(* CoDeSys 2.3 project: cy-wg-017-01.pro *)
(* Title: cy-wg-06 - ClevergyAS *)
(* Author: Andrea Ravasio *)
(* Libraries: Standard.lib 2.12.10 14:48:34, Util.lib 26.9.14 10:12:46, Visual.lib 2.12.10 14:48:34, WagoLibIdent.lib 25.2.13 11:12:16, WagoLibStatus.lib 2.12.10 14:48:32, SysLibFile.lib 2.12.10 14:48:34, SysLibRtc.lib 2.12.10 14:48:32, SysLibSockets.lib 10.2.11 09:20:54, SysLibEvent.lib 2.12.10 14:48:34, SysLibPlcCtrl.lib 2.12.10 14:48:32, SysLibCallback.lib 2.12.10 14:48:32, mod_com.lib 2.12.10 14:48:32, SerComm.lib 31.5.11 08:54:36, Serial_Interface_01.lib 22.4.13 12:50:14, Modb_l05.lib 22.4.13 12:50:12, Ethernet.lib 2.12.10 14:48:32, MBus_03.lib 22.7.15 16:25:47, WagoLibModbus_IP_01.lib 24.7.13 15:05:58, WagoLibMBX_01.lib 20.3.12 16:32:40, LON_01.lib 22.7.15 16:25:47 *)

(* PLC configuration (modules and I/O channels)
0750-9999/0545-0008 8 DO/DI Generic [Type_34_8_Channels] node 0, in %IB60 out %QB36 {INTTypePAAssignment = PLC; INTTypeModule = plugged}
  VPN_ST2 AT %IX30.0 [BOOLOnX_I] Ch_1 Digital input
  LAMP_AL AT %QX18.0 [BOOLOnX_Q] Ch_1 Digital output
  KEY_QE_ST AT %IX30.1 [BOOLOnX_I] Ch_2 Digital input
  CIR02_EN AT %QX18.1 [BOOLOnX_Q] Ch_2 Digital output
  CTL01_ST AT %IX30.2 [BOOLOnX_I] Ch_3 Digital input
  CIR01_EN AT %QX18.2 [BOOLOnX_Q] Ch_3 Digital output
  CTL02_ST AT %IX30.3 [BOOLOnX_I] Ch_4 Digital input
  AT %QX18.3 [BOOLOnX_Q] Ch_4 Digital output
  CIRD01_A_AL AT %IX30.4 [BOOLOnX_I] Ch_5 Digital input
  AT %QX18.4 [BOOLOnX_Q] Ch_5 Digital output
  CIRD01_A_AUTO AT %IX30.5 [BOOLOnX_I] Ch_6 Digital input
  AT %QX18.5 [BOOLOnX_Q] Ch_6 Digital output
  CIRD01_B_AL AT %IX30.6 [BOOLOnX_I] Ch_7 Digital input
  AT %QX18.6 [BOOLOnX_Q] Ch_7 Digital output
  CIRD01_B_AUTO AT %IX30.7 [BOOLOnX_I] Ch_8 Digital input
  AT %QX18.7 [BOOLOnX_Q] Ch_8 Digital output
0750-9999/0400-0008 8 DI Generic [Type_1_8_Channels] node 1, in %IB60 out %QB36 {INTTypePAAssignment = PLC; INTTypeModule = plugged}
  CIRD02_A_AL AT %IX30.8 [BOOLOnX_I] I 1: Digital Input
  CIR03_AL AT %IX30.9 [BOOLOnX_I] I 2: Digital Input
  CIRD02_A_AUTO AT %IX30.10 [BOOLOnX_I] I 3: Digital Input
  CIR03_AUTO AT %IX30.11 [BOOLOnX_I] I 4: Digital Input
  CIRD02_B_AL AT %IX30.12 [BOOLOnX_I] I 5: Digital Input
  CIR02_AL AT %IX30.13 [BOOLOnX_I] I 6: Digital Input
  CIRD02_B_AUTO AT %IX30.14 [BOOLOnX_I] I 7: Digital Input
  CIR02_ST AT %IX30.15 [BOOLOnX_I] I 8: Digital Input
0750-9999/0400-0004 4 DI Generic [Type_1_4_Channels] node 2, in %IB61 out %QB37 {INTTypePAAssignment = PLC; INTTypeModule = plugged}
  CIR02_AUTO AT %IX31.0 [BOOLOnX_I] I 1: Digital Input
  CIR01_ST AT %IX31.1 [BOOLOnX_I] I 2: Digital Input
  CIR01_AL AT %IX31.2 [BOOLOnX_I] I 3: Digital Input
  CIR01_AUTO AT %IX31.3 [BOOLOnX_I] I 4: Digital Input
0750-0478 2 AI 0-10V 16 Bit S.E. [Type_8_2_Channels] node 3, in %IB56 out %QB36 {INTTypePAAssignment = PLC; INTTypeModule = plugged}
  VRD04_ST AT %IW0 [WORDOnW_I] I 1: Analog Input
  VRD05_ST AT %IW1 [WORDOnW_I] I 2: Analog Input
0753-0648 LON-FTT [Type_55_1_Channels] node 4, in %IB56 out %QB36 {INTTypePAAssignment = PLC; INTTypeModule = plugged; DataStream = .; DataStream = .; DataStream = .; DataStream = .; DataStream = .; DataStream = .; DataStream = .; DataStream = .; DataStream = .; DataStream = .; DataStream = .; DataStream = .; DataStream = .; DataStream = .; DataStream = .; DataStream = .; DataStream = .; DataStream = .; DataStream = .; DataStream = .; DataStream = .; DataStream = .; DataStream = .; DataStream = .; DataStream = .; DataStream = .; DataStream = .; DataStream = .; DataStream = .; DataStream = .; DataStream = .; DataStream = .; DataStream = .; DataStream = .; DataStream = .; DataStream = .; DataStream = .; DataStream = .; DataStream = .; DataStream = .; DataStream = .; DataStream = .; DataStream = .; DataStream = .; DataStream = .; DataStream = .; DataStream = .; DataStream = .; DataStream = .; DataStream = .; DataStream = .; DataStream = .; DataStream = .; DataStream = .; DataStream = .; DataStream = .; DataStream = .; DataStream = .; DataStream = .; DataStream = .; DataStream = .; DataStream = .; DataStream = .; DataStream = .; DataStream = .; DataStream = .; DataStream = .; DataStream = .; DataStream = .; DataStream = .; DataStream = .; DataStream = .; DataStream = .; DataStream = .; DataStream = .; DataStream = .; DataStream = .; DataStream = .; DataStream = .; DataStream = .; DataStream = .; DataStream = .; DataStream = .; DataStream = .; DataStream = .; DataStream = .; DataStream = .; DataStream = .; DataStream = .; DataStream = .; DataStream = .; DataStream = .; DataStream = .; DataStream = .; DataStream = .; DataStream = .; DataStream = .; DataStream = .; DataStream = .; DataStream = .; DataStream = .; DataStream = .; DataStream = .; DataStream = .; DataStream = .; DataStream = .; DataStream = .; DataStream = .; DataStream = .; DataStream = .; DataStream = .; DataStream = .; DataStream = .; DataStream = .; DataStream = .; DataStream = .; DataStream = .; DataStream = .; DataStream = .; DataStream = .; DataStream = .; DataStream = .; DataStream = .; DataStream = .; DataStream = .; DataStream = .; DataStream = .; DataStream = .; DataStream = .; DataStream = .; DataStream = .; DataStream = .; DataStream = .; DataStream = .; DataStream = .; DataStream = .; DataStream = .; DataStream = .; DataStream = .; DataStream = .; DataStream = .; DataStream = .; DataStream = .; DataStream = .; DataStream = .; DataStream = .; DataStream = .; DataStream = .; DataStream = .; DataStream = .; DataStream = .; DataStream = .; DataStream = .; DataStream = .; DataStream = .; DataStream = .; DataStream = .; DataStream = .; DataStream = .; DataStream = .; DataStream = .; DataStream = .; DataStream = .; DataStream = .; DataStream = .; DataStream = .; DataStream = .; DataStream = .; DataStream = .; DataStream = .; DataStream = .; DataStream = .; DataStream = .; DataStream = .; DataStream = .; DataStream = .; DataStream = .; DataStream = .; DataStream = .; DataStream = .; DataStream = .; DataStream = .; DataStream = .; DataStream = .; DataStream = .; DataStream = .; DataStream = .; DataStream = .; DataStream = .; DataStream = .; DataStream = .; DataStream = .; DataStream = .; DataStream = .; DataStream = .; DataStream = .; DataStream = .; DataStream = .; DataStream = .; DataStream = .}
  AT %IB4 [BYTEOnB_I] First Byte of 24
  AT %QB0 [BYTEOnB_Q] First Byte of 24
0750-0464#04 2/4 AI RTD / ADJ./ HA [Type_44_4_Channels] node 5, in %IB60 out %QB36 {INTTypePAAssignment = PLC; INTTypeModule = plugged}
  S01 AT %IW14 [INTOnW_I] Channel 1
  S02 AT %IW15 [INTOnW_I] Channel 2
  S03 AT %IW16 [INTOnW_I] Channel 3
  S04 AT %IW17 [INTOnW_I] Channel 4
0750-0464#04 2/4 AI RTD / ADJ./ HA [Type_44_4_Channels] node 6, in %IB84 out %QB60 {INTTypePAAssignment = PLC; INTTypeModule = plugged}
  S05 AT %IW18 [INTOnW_I] Channel 1
  S07 AT %IW19 [INTOnW_I] Channel 2
  S06 AT %IW20 [INTOnW_I] Channel 3
  S08 AT %IW21 [INTOnW_I] Channel 4
0750-0556 2 AO ±10V [Type_14_2_Channels] node 7, in %IB92 out %QB60 {INTTypePAAssignment = PLC; INTTypeModule = plugged}
  VRD04_CTRL AT %QW12 [WORDOnW_Q] O 1: Analog Output
  VRD05_CTRL AT %QW13 [WORDOnW_Q] O 2: Analog Output
0750-0650/0003-0000#03 RS 232 C Interface (Adjustable), 3 Byte [Type_21_1_Channels] node 8, in %IB100 out %QB60 {INTTypePAAssignment = PLC; INTTypeModule = plugged}
  AT %IX22.0 [BOOLOnX_I] Transmission acknowledgement
  AT %IX22.1 [BOOLOnX_I] Reception request
  AT %IX22.2 [BOOLOnX_I] Initialization acknowledgement
  AT %IX22.3 [BOOLOnX_I] Input buffer is full
  AT %IX22.4 [BOOLOnX_I] Number of received characters Bit 0
  AT %IX22.5 [BOOLOnX_I] Number of received characters Bit 1
  AT %IX22.6 [BOOLOnX_I] Number of received characters Bit 2
  AT %IB45 [BYTEOnB_I] Input data Byte 0
  AT %IB46 [BYTEOnB_I] Input data Byte 1
  AT %IB47 [BYTEOnB_I] Input data Byte 2
  AT %QX14.0 [BOOLOnX_Q] Transmission request
  AT %QX14.1 [BOOLOnX_Q] Reception acknowledgement
  AT %QX14.2 [BOOLOnX_Q] Initialization request
  AT %QX14.4 [BOOLOnX_Q] Number of characters Bit 0
  AT %QX14.5 [BOOLOnX_Q] Number of characters Bit 1
  AT %QX14.6 [BOOLOnX_Q] Number of characters Bit 2
  AT %QB29 [BYTEOnB_Q] Output data Byte 0
  AT %QB30 [BYTEOnB_Q] Output data Byte 1
  AT %QB31 [BYTEOnB_Q] Output data Byte 2
0750-0653/0003-0000#03 RS485 Interface (Adjustable), 3 Bytes [Type_21_1_Channels] node 9, in %IB100 out %QB64 {INTTypePAAssignment = PLC; INTTypeModule = plugged}
  AT %IX24.0 [BOOLOnX_I] Transmission acknowledgement
  AT %IX24.1 [BOOLOnX_I] Reception request
  AT %IX24.2 [BOOLOnX_I] Initialization acknowledgement
  AT %IX24.3 [BOOLOnX_I] Input buffer is full
  AT %IX24.4 [BOOLOnX_I] Number of received characters Bit 0
  AT %IX24.5 [BOOLOnX_I] Number of received characters Bit 1
  AT %IX24.6 [BOOLOnX_I] Number of received characters Bit 2
  AT %IB49 [BYTEOnB_I] Input data Byte 0
  AT %IB50 [BYTEOnB_I] Input data Byte 1
  AT %IB51 [BYTEOnB_I] Input data Byte 2
  AT %QX16.0 [BOOLOnX_Q] Transmission request
  AT %QX16.1 [BOOLOnX_Q] Reception acknowledgement
  AT %QX16.2 [BOOLOnX_Q] Initialization request
  AT %QX16.4 [BOOLOnX_Q] Number of characters Bit 0
  AT %QX16.5 [BOOLOnX_Q] Number of characters Bit 1
  AT %QX16.6 [BOOLOnX_Q] Number of characters Bit 2
  AT %QB33 [BYTEOnB_Q] Output data Byte 0
  AT %QB34 [BYTEOnB_Q] Output data Byte 1
  AT %QB35 [BYTEOnB_Q] Output data Byte 2
0750-0461/0000-0007 2 AI PT100 Resistor Measur. 10R-5k0 [Type_8_2_Channels] node 10, in %IB104 out %QB68 {INTTypePAAssignment = PLC; INTTypeModule = plugged}
  VRD01_ST AT %IW26 [WORDOnW_I] I 1: Analog Input
  VRD02_ST AT %IW27 [WORDOnW_I] I 2: Analog Input
0750-0461/0000-0007 2 AI PT100 Resistor Measur. 10R-5k0 [Type_8_2_Channels] node 11, in %IB108 out %QB72 {INTTypePAAssignment = PLC; INTTypeModule = plugged}
  VRD03_ST AT %IW28 [WORDOnW_I] I 1: Analog Input
  AT %IW29 [WORDOnW_I] I 2: Analog Input
0750-9999/0500-0002 2 DO Generic [Type_10_2_Channels] node 12, in %IB62 out %QB37 {INTTypePAAssignment = PLC; INTTypeModule = plugged}
  VRD01_OP AT %QX18.8 [BOOLOnX_Q] O 1: Digital Output
  VRD01_CL AT %QX18.9 [BOOLOnX_Q] O 2: Digital Output
0750-9999/0500-0002 2 DO Generic [Type_10_2_Channels] node 13, in %IX31.4 out %QB37 {INTTypePAAssignment = PLC; INTTypeModule = plugged}
  VRD02_OP AT %QX18.10 [BOOLOnX_Q] O 1: Digital Output
  VRD02_CL AT %QX18.11 [BOOLOnX_Q] O 2: Digital Output
0750-9999/0500-0002 2 DO Generic [Type_10_2_Channels] node 14, in %IX31.4 out %QX18.10 {INTTypePAAssignment = PLC; INTTypeModule = plugged}
  VRD03_OP AT %QX18.12 [BOOLOnX_Q] O 1: Digital Output
  VRD03_CL AT %QX18.13 [BOOLOnX_Q] O 2: Digital Output
Fieldbus variables [FB_VARS] node 1, in %IB0 out %QB0
Flag variables [FLAG_VARS] node 2, in %IB0 out %QB0
Modbus-Master [MB_MASTER] node 3, in %IB0 out %QB0
*)

(* Global variable list: Global_Constants *)
VAR_GLOBAL CONSTANT

	Plant_NAME			: STRING :='cySN:17 cyVER:1 - ';
	Plant_SN			: DWORD  :=17;	(* S/N Impianto di telecontrollo *)
	Plant_SW_VER		: WORD   :=1;		(* Versione SW installata *)


	(* Colour defines *)
	COLOR_RED			: DWORD	:= 16#2020F0;
	COLOR_YELLOW		: DWORD	:= 16#20F0F0;
	COLOR_GREEN			: DWORD	:= 16#20F020;
	COLOR_LIGHT_GREEN	: DWORD := 16#006000;

	(* Parameters *)
	Plant_DefaultTAmb	: INT	:=100;		(* [.1°C] Temperatura ambiente di default in caso di rottura sonda *)
	Plant_MaxRunTAmb	: INT   :=250; 		(* [.1°C] Temperatura ambiente massima funzionamento impianto *)
	Plant_AntiFreezeTAmb: INT   :=-40;		(* [.1°C] Antifreeze temperature, start circulators *)
	Plant_VRD_TAlarm	: INT   :=450; 		(* [.1°C] Temperatura di allarme VRD, blocco *)
	Plant_VRD_TMax		: INT   :=430; 		(* [.1°C] Setpoint massimo per uscita VRD *)
	Plant_VRD_TDefault	: INT	:=300;		(* [.1°C] Temperatura di default in caso di errore climatica *)
	Plant_CirOffDelay	: TIME	:=T#30m;	(* (Def.T#15m) Ritardo spegnimento pompe per ricircolo caldaia *)
	Plant_CirOnDelay	: TIME	:=T#15m;
	Plant_MaxWaterLoss	: WORD  :=2;		(* [lt/h] Massima perdita del circuito *)

	(* Filesystem *)
	FilesPath  			: STRING :='S:\';

	(* TCP Logger *)
	Logger_SERVER		: STRING:='';
	Logger_IP			: STRING:='192.168.100.3';
	Logger_PORT			: WORD  :=80;
	Logger_GETSTART		: STRING:='GET /cygmsrv/hsgm.ashx?';
	Logger_GETEND		: STRING:='$R$N$R$N';
	Logger_CHECK		: STRING:='True';
	Logger_CRLF			: STRING:='$R$N';
	Logger_DataFile		: STRING:='S:\LOG.DAT';
	Logger_DataFileOld	: STRING:='S:\LOG.BCK';
	Logger_IndexFile	: STRING:='S:\LOG.IDX';
	Logger_ConnRetries	: BYTE:=5;
	Logger_RecoverMsgs	: BYTE:=25;

	(* TCP Remote *)
	Remote_PORT			: WORD  :=10;
	Remote_WELCOME		: STRING:='Connected$R$N';
	Remote_OK			: STRING:='OK$R$N';
	Remote_ERROR		: STRING:='ERROR$R$N';

	(* TCP Sockets *)
	MAX_SEND_TCP_SERVER					 : DWORD:=3000;(*60000*)
	MAX_RECEIVE_TCP_SERVER				 : DWORD:=3000;
	MAX_RECEIVE_TCP_SERVER_SOCKET	 	 : DWORD:=1500;
	MAX_SEND_TCP_CLIENT					 : DWORD:=3000;(*15000*)
	MAX_RECEIVE_TCP_CLIENT				 : DWORD:=1500;
	MAX_RECEIVE_TCP_CLIENT_SOCKET		 : DWORD:=1500;
	MAX_RECEIVE_UDP_SERVER				 : INT  :=1472;
	MAX_RECEIVE_UDP_CLIENT				 : INT  :=1472;
	CONNECT_WATCHDOG_TIME				 : TIME :=t#10s;

END_VAR

(* Global variable list: Global_Retain *)
VAR_GLOBAL RETAIN PERSISTENT
	Mode_Manual : BOOL := FALSE;

	GRU01_Clima	: typ_Clima;

	VRD01_Clima : typ_Clima;
	VRD02_Clima : typ_Clima;
	VRD03_Clima : typ_Clima;
	VRD04_Clima : typ_Clima;
	VRD05_Clima : typ_Clima;

	Ctl01_Counter	:	DWORD;
	Ctl02_Counter	:	DWORD;

END_VAR

(* Global variable list: Global_Variables *)
VAR_GLOBAL

	SYS    : typ_SYS;
	Logger : typ_Logger;

	Lamp	:	PLANT_STATUS;
	T_AMB	:	INT;		(* Environment temperature *)

	(**** PLANT OBJECTS ****)
	(*...*)
	GRU01	:	obj_CAL_VT300GW2 := (ID:=1);

	(* Water counter (NB il peso è moltiplicato per 10) *)
	CTL01	:	obj_CTL	:= (ID:=1, Peso:=10);	(* Domestic water *)
	CTL02	:	obj_CTL	:= (ID:=2, Peso:=10);	(* Compensation *)

	(* Heat counter *)
	CTB01	:	obj_MBUS_CTB_SHARKY775 := (ID:=1, Address:=1);
	CTB02	:	obj_MBUS_CTB_SHARKY775 := (ID:=2, Address:=2);

	(* Cronothermostat *)
	THER01	:	obj_CRONTER := (ID:=1, Local_MaxRunTAmb:=250);
	THER02	:	obj_CRONTER := (ID:=2, Local_MaxRunTAmb:=250);
	THER03	:	obj_CRONTER := (ID:=3, Local_MaxRunTAmb:=250);
	THER04	:	obj_CRONTER := (ID:=4, Local_MaxRunTAmb:=250);
	THER05	:	obj_CRONTER := (ID:=5, Local_MaxRunTAmb:=250);

	CronEd	: 	obj_CRON_EDITOR;

	(* Pump *)
	CIR01	:	obj_CIR	:= (ID:=1, OnDelay:=T#1m);
	CIR02	:	obj_CIR	:= (ID:=2, OnDelay:=T#1m);

	(* ModBus Pumps *)
	CIR03	:	obj_MODBUS_CIR := (ID:=1, Address:=1, OnDelay:=T#1m);

	(* Modbus double pumps *)
	CIRD01	:	obj_MODBUS_CIR_DOPPIO_new := (ID:=1, Address1:=2, Address2:=3, OnDelay:=T#1m);
	CIRD02	:	obj_MODBUS_CIR_DOPPIO_new := (ID:=2, Address1:=4, Address2:=5, OnDelay:=T#1m);

	(* Valves *)
	VRD01	:	obj_VRD_POT	:= (ID:=1);
	VRD02	:	obj_VRD_POT	:= (ID:=2);
	VRD03	:	obj_VRD_POT	:= (ID:=3);

	VRD04	:	obj_VRD 	:= (ID:=4, ReducedRange := FALSE);
	VRD05	:	obj_VRD 	:= (ID:=5, ReducedRange := FALSE);

	(* Temperature probes *)
	TPV01	:	obj_TPV := (ID:=1);
	TPV02	:	obj_TPV := (ID:=2, IN_WMIN:=50 , IN_WMAX:=800);
	TPV03	:	obj_TPV := (ID:=3, IN_WMIN:=50 , IN_WMAX:=800);
	TPV04	:	obj_TPV := (ID:=4);
	TPV05	:	obj_TPV := (ID:=5);
	TPV06	:	obj_TPV := (ID:=6);
	TPV07	:	obj_TPV := (ID:=7);
	TPV08	:	obj_TPV := (ID:=8);

	(* Zigbee temperature probes *)
	ZTHL09	:	obj_ZTHL := (ID:=1, Address:=1);
	ZTHL10	:	obj_ZTHL := (ID:=2, Address:=2);
	ZTHL11	:	obj_ZTHL := (ID:=3, Address:=3);
	ZTHL12	:	obj_ZTHL := (ID:=4, Address:=4);
	ZTHL13	:	obj_ZTHL := (ID:=5, Address:=5);
	ZTHL14	:	obj_ZTHL := (ID:=6, Address:=6);

	(** Communication **)
	(* ModBus *)
	MODB01	:	obj_MODBUS		:= (ID:=1, COM:=3, BAUDRATE:=BAUD_9600, RS485:=TRUE);
	MODB02	:	obj_MODBUS_TCP 	:= (ID:=1, IP:='192.168.100.11');

	(* M-Bus *)
	MBUS01	:	obj_MBUS		:= (ID:=1, COM:=2, BAUDRATE:=BAUD_2400);

	(**** SIMULATION ONLY ****)
	(*...*)
END_VAR

(* Global variable list: LON/Module_1/InterfaceBlock_Module_1 *)
VAR_GLOBAL CONSTANT
(******************************************)
(* Automatic generated code, do not edit! *)
(******************************************)
	abSignature_Module_1 : ARRAY[0..15] OF BYTE := 16#7A,16#26,16#60,16#DB,16#56,16#3B,16#16,16#40,16#89,16#16,16#11,16#E4,16#B0,16#D6,16#83,16#3B;
	wConfigSize_Module_1 : WORD := 504;
	abInterface_Module_1 : ARRAY[0..125] OF DWORD :=
		16#1028C19F, 16#2137A508, 16#6041B800, 16#06246830, 16#428B2E71, 16#64B95263, 16#FE000902, 16#2A050140, 
		16#201E4092, 16#8BD6B010, 16#8102570F, 16#1890E46A, 16#5C1D0704, 16#D47157C7, 16#1D2B759C, 16#539D1D5A, 
		16#8D25581D, 16#286C1D4F, 16#65AAA48D, 16#A999312F, 16#3871E72B, 16#2E679A2C, 16#1526509A, 16#A942353A, 
		16#2CD9B76E, 16#AA15FBB4, 16#4EBA63CB, 16#244B36E8, 16#BA6FF382, 16#3B16A4DC, 16#65DBB67D, 16#16245DB7, 
		16#CBCA2D8B, 16#AE5B9800, 16#96959AD6, 16#DCB275E3, 16#980083EE, 16#D22A265F, 16#96EED4B7, 16#E6D6A51B, 
		16#B49229B9, 16#659BD6E8, 16#922C6495, 16#A68DAF9A, 16#146D324C, 16#0BF59CD9, 16#F0E6207B, 16#A95A0509, 
		16#0C30595F, 16#2A0F6A98, 16#1548A5A5, 16#2835283B, 16#CA0DCB36, 16#138125DA, 16#9097AD54, 16#7A002B99, 
		16#0E1D8A54, 16#A3A65F63, 16#E7C47284, 16#CB52452D, 16#EC15B86D, 16#A99847E4, 16#04176EDD, 16#5C8A4C1D, 
		16#1C5445A1, 16#988C80B5, 16#45CDF448, 16#437D14CF, 16#1908420B, 16#29D10D87, 16#8F957715, 16#BA63838A, 
		16#358C6C0D, 16#DCA67D0B, 16#50958048, 16#0943D4E8, 16#1BD66D51, 16#870EB015, 16#3DA1A3F2, 16#51472006, 
		16#6AD45591, 16#AD028665, 16#09DCFECE, 16#00010604, 16#EE3FC081, 16#1B047261, 16#4C28E600, 16#38E51802, 
		16#ED3602AC, 16#1EAC8339, 16#837136A7, 16#3520E7F4, 16#E020C09F, 16#2340A3D3, 16#88B153A1, 16#08783AC0, 
		16#784A0804, 16#5A040428, 16#0DD83178, 16#0133084F, 16#6B86E1E9, 16#28AE2588, 16#1AB2B876, 16#8E6B0BE3, 
		16#E640AE29, 16#E41A23B9, 16#41946BCD, 16#B9F658AE, 16#91E6DA84, 16#AE519B6B, 16#F5B95675, 16#6B58E8DA, 
		16#95AE65A3, 16#DA66BA66, 16#AA6B1AEA, 16#F601AC75, 16#4082302E, 16#8CE93226, 16#F2000AEC, 16#03C62483, 
		16#2FC18102, 16#6E076B52, 16#508B3BAD, 16#8F683131, 16#C1D66193, 16#2056FDCE;
END_VAR

(* Global variable list: LON/Module_1/Runtime_Module_1 *)
VAR_GLOBAL
(******************************************)
(* Automatic generated code, do not edit! *)
(******************************************)
	mbxModule_1 : MBX_Full;
	InDataTelegram_Module_1 : ARRAY[0..255] OF BYTE;
	OutDataTelegram_Module_1 : ARRAY[0..511] OF BYTE;

	xInitRunning_Module_1 : BOOL := FALSE;
	unLastLen_mbxModule_1 : UINT;
END_VAR

(* Data type in LON/Enumerations *)
TYPE alarm_type_t :
(
	AL_HEADER := -13,
	AL_FOOTER := -12,
	AL_DEBUG := -11,
	AL_INFO := -10,
	AL_SYSTEM_INFO := -6,
	AL_VALUE_INVALID := -5,
	AL_CONSTANT := -4,
	AL_OFFLINE := -3,
	AL_UNKNOWN := -2,
	AL_NUL := -1,
	AL_NO_CONDITION := 0,
	AL_ALM_CONDITION := 1,
	AL_TOT_SVC_ALM_1 := 2,
	AL_TOT_SVC_ALM_2 := 3,
	AL_TOT_SVC_ALM_3 := 4,
	AL_LOW_LMT_CLR_1 := 5,
	AL_LOW_LMT_CLR_2 := 6,
	AL_HIGH_LMT_CLR_1 := 7,
	AL_HIGH_LMT_CLR_2 := 8,
	AL_LOW_LMT_ALM_1 := 9,
	AL_LOW_LMT_ALM_2 := 10,
	AL_HIGH_LMT_ALM_1 := 11,
	AL_HIGH_LMT_ALM_2 := 12,
	AL_FIR_ALM := 13,
	AL_FIR_PRE_ALM := 14,
	AL_FIR_TRBL := 15,
	AL_FIR_SUPV := 16,
	AL_FIR_TEST_ALM := 17,
	AL_FIR_TEST_PRE_ALM := 18,
	AL_FIR_ENVCOMP_MAX := 19,
	AL_FIR_MONITOR_COND := 20,
	AL_FIR_MAINT_ALERT := 21,
	AL_FATAL_ERROR := 30,
	AL_ERROR := 31,
	AL_WARNING := 32
);
END_TYPE

(* Data type in Logger *)
TYPE en_Logger_ErrLev :
(
	EL_Log			:=0,
	EL_Wrn			:=1,
	EL_Alarm		:=2,
	EL_AlarmStop	:=3
);
END_TYPE

(* Data type in Logger *)
TYPE en_Logger_Status :
(
	S_Logger_UNKNOWN := 0,
	S_Logger_IDLE,
	S_Logger_WAITCONN,
	S_Logger_WAITTX,
	S_Logger_WAITRESP,
	S_Logger_ERROR
);
END_TYPE

(* Data type *)
TYPE en_SYS_Objects :
(
	EO_SYS		:=0,  (* PLC *)
	EO_VPN		:=1,  (* VPN *)
	EO_DOOR		:=2,  (* Door & access control *)

	EO_CAL		:=10, (* Caldaia *)
	EO_CIR		:=11, (* Circolatore *)
	EO_CRON		:=12, (* Crono-termostato *)
	EO_VRD		:=13, (* Valvola miscelatore pannelli *)
	EO_CTL		:=14, (* Contalitri *)
	EO_CTB		:=15, (* Contabilizzatore *)
	EO_TPV		:=16, (* Temperature probes values *)
	EO_PPV		:=17, (* Pressure probes values *)
	EO_PBV		:=18, (* Over-Pressure Alarms *)
	EO_TBV		:=19, (* Over-Temperature Alarms *)
	EO_PMV		:=20, (* Under-Pressure Alarms *)
	EO_GRU		:=21, (* Gruppo termico *)
	EO_PDC		:=22, (* Pompa di calore *)
	EO_SOL		:=23, (* Pannello solare termico *)
	EO_ESOL		:=24, (* Pannello solare fotovoltaico *)
	EO_GAS		:=25, (* Contatore GAS *)
	EO_PORT		:=26, (* Misuratore di portata *)
	EO_FPV		:=27, (* Flow probes values *)
	EO_ANZ		:=28, (* Analizzatore di rete *)
	EO_SCA		:=29, (* Signal Control Alarms *)
	EO_LUX		:=30, (* Base Illumination point *)
	EO_LUXM		:=31, (* Metered Illumination point *)
	EO_PSG		:=32, (* Sensore di passaggio *)
	EO_HVAC		:=33, (* Heating, Ventilating and Air Conditioning *)
	EO_HYGRV	:=34, (* Relative Humidity sensors value *)
	EO_COOV		:=35, (* Carbon Dioxide CO2 sensors value *)
	EO_INV		:=36, (* Inverter *)
	EO_STR		:=37, (* Smart string box *)

	EO_CIRD		:=39, (* Double CIR *)
	EO_ACS		:=40, (* Hot domestic water *)
	EO_FRG		:=41, (* Frigo *)
	EO_THER		:=42, (* Thermostat *)

	EO_ZGW			:=200,  (* ZigBee - Gateway *)
	EO_ZRM			:=201,	(* ZigBee - Repeater *)
	EO_ZREL			:=202,	(* ZigBee - Actuator rele *)
	EO_ZTHL			:=203,	(* ZigBee - Temperature Sensor *)

	EO_ASGW			:=250,	(* ASi - Gateway *)
	EO_ASCBI		:=251,	(* ASi - Input Board, Ciabatta *)

	EO_LON			:=1000, (* Bus - LON *)
	EO_MODBUS		:=1001, (* Bus - MODBUS *)
	EO_MBUS			:=1002, (* Bus - M-BUS *)
	EO_MODBUS_TCP	:=1003, (* Bus - MODBUS TCP *)

	EO_GENERIC		:=9000, (* Generic dataset *)
	EO_EXPO			:=9001 (* EXPO dataset *)
);
END_TYPE

(* Data type *)
TYPE en_SYS_Status :
(
	S_UNKNOWN  := 0,
	S_STARTUP,
	S_INIT_RTC,
	S_INIT_VAR,
	S_AUTOTEST,
	S_RUNNING,
	S_SHUTDOWN,
	S_HALT
);
END_TYPE

(* Data type in LON/Enumerations *)
TYPE file_request_t :
(
	FR_NUL := -1,
	FR_OPEN_TO_SEND := 0,
	FR_OPEN_TO_RECEIVE := 1,
	FR_CLOSE_FILE := 2,
	FR_CLOSE_DELETE_FILE := 3,
	FR_DIRECTORY_LOOKUP := 4,
	FR_OPEN_TO_SEND_RA := 5,
	FR_OPEN_TO_RECEIVE_RA := 6
);
END_TYPE

(* Data type in LON/Enumerations *)
TYPE file_status_t :
(
	FS_NUL := -1,
	FS_XFER_OK := 0,
	FS_LOOKUP_OK := 1,
	FS_OPEN_FAIL := 2,
	FS_LOOKUP_ERR := 3,
	FS_XFER_UNDERWAY := 4,
	FS_IO_ERR := 5,
	FS_TIMEOUT_ERR := 6,
	FS_WINDOW_ERR := 7,
	FS_AUTH_ERR := 8,
	FS_ACCESS_UNAVAIL := 9,
	FS_SEEK_INVALID := 10,
	FS_SEEK_WAIT := 11
);
END_TYPE

(* Data type in LON/Enumerations *)
TYPE hvac_t :
(
	HVAC_NUL := -1,
	HVAC_AUTO := 0,
	HVAC_HEAT := 1,
	HVAC_MRNG_WRMUP := 2,
	HVAC_COOL := 3,
	HVAC_NIGHT_PURGE := 4,
	HVAC_PRE_COOL := 5,
	HVAC_OFF := 6,
	HVAC_TEST := 7,
	HVAC_EMERG_HEAT := 8,
	HVAC_FAN_ONLY := 9,
	HVAC_FREE_COOL := 10,
	HVAC_ICE := 11,
	HVAC_MAX_HEAT := 12,
	HVAC_ECONOMY := 13,
	HVAC_DEHUMID := 14,
	HVAC_CALIBRATE := 15,
	HVAC_EMERG_COOL := 16,
	HVAC_EMERG_STEAM := 17,
	HVAC_MAX_COOL := 18,
	HVAC_HVC_LOAD := 19,
	HVAC_NO_LOAD := 20
);
END_TYPE

(* Data type in LON/Enumerations *)
TYPE object_request_t :
(
	RQ_NUL := -1,
	RQ_NORMAL := 0,
	RQ_DISABLED := 1,
	RQ_UPDATE_STATUS := 2,
	RQ_SELF_TEST := 3,
	RQ_UPDATE_ALARM := 4,
	RQ_REPORT_MASK := 5,
	RQ_OVERRIDE := 6,
	RQ_ENABLE := 7,
	RQ_RMV_OVERRIDE := 8,
	RQ_CLEAR_STATUS := 9,
	RQ_CLEAR_ALARM := 10,
	RQ_ALARM_NOTIFY_ENABLED := 11,
	RQ_ALARM_NOTIFY_DISABLED := 12,
	RQ_MANUAL_CTRL := 13,
	RQ_REMOTE_CTRL := 14,
	RQ_PROGRAM := 15,
	RQ_CLEAR_RESET := 16,
	RQ_RESET := 17,
	RQ_CLEAR_LOG := 18,
	RQ_LOAD_PROGRAM := 19,
	RQ_RUN_PROGRAM := 20,
	RQ_HALT_PROGRAM := 21,
	RQ_RESTART_PROGRAM := 22,
	RQ_UNLOAD_PROGRAM := 23,
	RQ_STEP_PROGRAM := 24
);
END_TYPE

(* Data type in LON/Enumerations *)
TYPE priority_level_t :
(
	PR_NUL := -1,
	PR_LEVEL_0 := 0,
	PR_LEVEL_1 := 1,
	PR_LEVEL_2 := 2,
	PR_LEVEL_3 := 3,
	PR_1 := 4,
	PR_2 := 5,
	PR_3 := 6,
	PR_4 := 7,
	PR_6 := 8,
	PR_8 := 9,
	PR_10 := 10,
	PR_16 := 11
);
END_TYPE

(* Data type in Plant_Objects *)
TYPE typ_Clima : (* CURVA CLIMATICA *)
STRUCT
	InitOK:		BOOL;
	Points: 	ARRAY [0..10] OF POINT;
END_STRUCT
END_TYPE

(* Data type in Plant_Objects *)
TYPE typ_Cron_Calendar :
STRUCT
	Profile		: ARRAY[0..384] OF BYTE;
END_STRUCT
END_TYPE

(* Data type in Plant_Objects *)
TYPE typ_Cron_Jolly :
STRUCT
	Start		: DT;
	End			: DT;
	Temp		: WORD;
	Flags		: WORD; (* B0:Enabled B1..B15:Unused *)
END_STRUCT
END_TYPE

(* Data type in Plant_Objects *)
TYPE typ_Cron_Profile :
STRUCT
	Flags		: WORD;
	Setpoint	: ARRAY [0..95] OF WORD;
END_STRUCT
END_TYPE

(* Data type in Plant_Objects *)
TYPE typ_Frigo :
STRUCT
	Status	:	BOOL;		(* 0=OFF, 1=ON	*)
	Mode	:	BOOL;		(* 0=COLD, 1=HOT	*)

END_STRUCT
END_TYPE

(* Data type in Logger *)
TYPE typ_Logger :
STRUCT
	Status		: en_Logger_Status;

	SendReq		: BOOL;
	SendIdx		: DWORD;
	SendData	: ARRAY [0..MAX_SEND_TCP_CLIENT] OF BYTE;
	SendLen		: DINT;

	TData		: ARRAY [0..MAX_SEND_TCP_CLIENT] OF BYTE;
	TLen		: DINT;

	LastIdxPos	: DWORD;

	(* Temporary variables used by objects *)
	s1			: STRING(256);
	i1			: WORD;

END_STRUCT
END_TYPE

(* Data type in Plant_Objects *)
TYPE typ_MODBUS_CIR :
STRUCT
	PumpStatus		:	WORD;
	PumpFault		:	BOOL;
	PumpBoardTemp	:	INT;	(* Electonic board temperature  [°C] *)
	PumpVoltage		:	WORD;	(* Input voltage rms [V] *)
	PumpCurrent		:	WORD;	(* Output current [E-3 A]	*)
	PumpRPM			:	WORD;	(* Round per minute [rpm] *)
	PumpPower		:	WORD;	(* Power [W] *)
	PumpOpTime		:	DWORD;	(* Pump operating time [h] *)
	PumpHead		:	WORD;	(* [E-1 m] *)
	PumpFlow		:	WORD;	(* Extimated flow [E-1 m3/h] *)
	PumpLiqTemp		:	WORD;	(* Liquid temperature [°C] *)
	PumpAlarm		:	ARRAY [0..14] OF WORD;

END_STRUCT
END_TYPE

(* Data type in Plant_Objects *)
TYPE typ_MODBUS_VAR : (* Gestione parametri MODBUS *)
STRUCT
	SlaveAddress	: BYTE;
	FunCode			: BYTE;
	FunAddress		: WORD;
	Refresh_Time	: BYTE; (* 0:No refresh x:Refresh in seconds *)
	Refresh_Cnt		: BYTE; (* INTERNAL *)
	Variable		: POINTER TO WORD;
	Variable_Size	: BYTE;
	Variable_Mirror : WORD; (* INTERNAL [Force refresh on read variables when <>0] *)
END_STRUCT
END_TYPE

(* Data type *)
TYPE typ_SYS :
STRUCT
	Status			: en_SYS_Status;
	Warning			: BOOL;
	Alarm			: BOOL;
	AlarmStop		: BOOL;

	Time_LogString	: STRING;
	Time_Year		: WORD;
	Time_Month		: BYTE;
	Time_Day		: BYTE;

	Time_CT_DT		: DT;
	Time_CT_Day		: WORD;
	Time_CT_Quarter	: BYTE;

	LastLogs_Idx	: BYTE;
	LastLogs_Dat	: ARRAY[0..5] OF STRING;
	LastLogs_Msg	: ARRAY[0..5] OF STRING;

END_STRUCT
END_TYPE

(* Data type in Plant_Objects *)
TYPE typ_VisuStrutturaMbus :
STRUCT

	sdNodoPresente: STRING(16);
	sdEnergia: STRING(16);
	sdPotenza: STRING(16);
	sdVolume: STRING(16);
	sdFlow: STRING(16);
	sdTempIngresso: STRING(8);
	sdTempaUscita: STRING(8);
	sdTempDelta: STRING(8);

END_STRUCT
END_TYPE

(* Data type in LON/NetworkVariables *)
TYPE typSnvtAlarm : 
STRUCT
	abLocation : ARRAY[0..5] OF BYTE;
	wObjectId : WORD;
	bAlarmType : BYTE (* enum type alarm_type_t *);
	bPriorityLevel : BYTE (* enum type priority_level_t *);
	wIndexToSnvt : WORD;
	abValue : ARRAY[0..3] OF BYTE;
	wYear : WORD;
	bMonth : BYTE;
	bDay : BYTE;
	bHour : BYTE;
	bMinute : BYTE;
	bSecond : BYTE;
	wMillisecond : WORD;
	abAlarmLimit : ARRAY[0..3] OF BYTE;
	bStatusInformation : BYTE; (* bit allocation of bStatusInformation:
	bit 0: NVI update counter LSB
	bit 1: NVI update counter
	bit 2: NVI update counter
	bit 3: NVI update counter MSB
	bit 4: timeout for NVI occurs (MaxRcvTime expired)
	bit 5: reserved
	bit 6: reserved
	bit 7: force NVO update *)
	bInternalUseOnly : BYTE; (* Do not use this byte in your application! *)
END_STRUCT
END_TYPE

(* Data type in LON/NetworkVariables *)
TYPE typSnvtFilePos : 
STRUCT
	diRwPtr : DINT;
	wRwLength : WORD;
	bStatusInformation : BYTE; (* bit allocation of bStatusInformation:
	bit 0: NVI update counter LSB
	bit 1: NVI update counter
	bit 2: NVI update counter
	bit 3: NVI update counter MSB
	bit 4: timeout for NVI occurs (MaxRcvTime expired)
	bit 5: reserved
	bit 6: reserved
	bit 7: force NVO update *)
	bInternalUseOnly : BYTE; (* Do not use this byte in your application! *)
END_STRUCT
END_TYPE

(* Data type in LON/NetworkVariables *)
TYPE typSnvtFileReq : 
STRUCT
	bRequest : BYTE (* enum type file_request_t *);
	wIndex : WORD;
	wReceiveTimeout : WORD;
	abDestAddress : ARRAY[0..4] OF BYTE (* union declaration *);
	bAuthOn : BYTE;
	bPrioOn : BYTE;
	bStatusInformation : BYTE; (* bit allocation of bStatusInformation:
	bit 0: NVI update counter LSB
	bit 1: NVI update counter
	bit 2: NVI update counter
	bit 3: NVI update counter MSB
	bit 4: timeout for NVI occurs (MaxRcvTime expired)
	bit 5: reserved
	bit 6: reserved
	bit 7: force NVO update *)
	bInternalUseOnly : BYTE; (* Do not use this byte in your application! *)
END_STRUCT
END_TYPE

(* Data type in LON/NetworkVariables *)
TYPE typSnvtFileStatus : 
STRUCT
	bStatus : BYTE (* enum type file_status_t *);
	wNumberOfFiles : WORD;
	wSelectedFile : WORD;
	abAdr : ARRAY[0..21] OF BYTE (* union declaration *);
	bStatusInformation : BYTE; (* bit allocation of bStatusInformation:
	bit 0: NVI update counter LSB
	bit 1: NVI update counter
	bit 2: NVI update counter
	bit 3: NVI update counter MSB
	bit 4: timeout for NVI occurs (MaxRcvTime expired)
	bit 5: reserved
	bit 6: reserved
	bit 7: force NVO update *)
	bInternalUseOnly : BYTE; (* Do not use this byte in your application! *)
END_STRUCT
END_TYPE

(* Data type in LON/NetworkVariables *)
TYPE typSnvtHvacMode : 
STRUCT
	bSnvtHvacMode : BYTE (* enum type hvac_t *);
	bStatusInformation : BYTE; (* bit allocation of bStatusInformation:
	bit 0: NVI update counter LSB
	bit 1: NVI update counter
	bit 2: NVI update counter
	bit 3: NVI update counter MSB
	bit 4: timeout for NVI occurs (MaxRcvTime expired)
	bit 5: reserved
	bit 6: reserved
	bit 7: force NVO update *)
	bInternalUseOnly : BYTE; (* Do not use this byte in your application! *)
END_STRUCT
END_TYPE

(* Data type in LON/NetworkVariables *)
TYPE typSnvtObjRequest : 
STRUCT
	wObjectId : WORD;
	bObjectRequest : BYTE (* enum type object_request_t *);
	bStatusInformation : BYTE; (* bit allocation of bStatusInformation:
	bit 0: NVI update counter LSB
	bit 1: NVI update counter
	bit 2: NVI update counter
	bit 3: NVI update counter MSB
	bit 4: timeout for NVI occurs (MaxRcvTime expired)
	bit 5: reserved
	bit 6: reserved
	bit 7: force NVO update *)
	bInternalUseOnly : BYTE; (* Do not use this byte in your application! *)
END_STRUCT
END_TYPE

(* Data type in LON/NetworkVariables *)
TYPE typSnvtObjStatus : 
STRUCT
	wObjectId : WORD;
	bBitfieldByteOffset2 : BYTE (* bit field *);
	bBitfieldByteOffset3 : BYTE (* bit field *);
	bBitfieldByteOffset4 : BYTE (* bit field *);
	bBitfieldByteOffset5 : BYTE (* bit field *);
	bStatusInformation : BYTE; (* bit allocation of bStatusInformation:
	bit 0: NVI update counter LSB
	bit 1: NVI update counter
	bit 2: NVI update counter
	bit 3: NVI update counter MSB
	bit 4: timeout for NVI occurs (MaxRcvTime expired)
	bit 5: reserved
	bit 6: reserved
	bit 7: force NVO update *)
	bInternalUseOnly : BYTE; (* Do not use this byte in your application! *)
END_STRUCT
END_TYPE

(* Data type in LON/NetworkVariables *)
TYPE typSnvtState : 
STRUCT
	bBitfieldByteOffset0 : BYTE (* bit field *);
	bBitfieldByteOffset1 : BYTE (* bit field *);
	bStatusInformation : BYTE; (* bit allocation of bStatusInformation:
	bit 0: NVI update counter LSB
	bit 1: NVI update counter
	bit 2: NVI update counter
	bit 3: NVI update counter MSB
	bit 4: timeout for NVI occurs (MaxRcvTime expired)
	bit 5: reserved
	bit 6: reserved
	bit 7: force NVO update *)
	bInternalUseOnly : BYTE; (* Do not use this byte in your application! *)
END_STRUCT
END_TYPE

(* Data type in LON/NetworkVariables *)
TYPE typSnvtSwitch : 
STRUCT
	bValue : BYTE;
	siState : SINT;
	bStatusInformation : BYTE; (* bit allocation of bStatusInformation:
	bit 0: NVI update counter LSB
	bit 1: NVI update counter
	bit 2: NVI update counter
	bit 3: NVI update counter MSB
	bit 4: timeout for NVI occurs (MaxRcvTime expired)
	bit 5: reserved
	bit 6: reserved
	bit 7: force NVO update *)
	bInternalUseOnly : BYTE; (* Do not use this byte in your application! *)
END_STRUCT
END_TYPE

(* Data type in LON/NetworkVariables *)
TYPE typSnvtTempP : 
STRUCT
	iSnvtTempP : INT;
	bStatusInformation : BYTE; (* bit allocation of bStatusInformation:
	bit 0: NVI update counter LSB
	bit 1: NVI update counter
	bit 2: NVI update counter
	bit 3: NVI update counter MSB
	bit 4: timeout for NVI occurs (MaxRcvTime expired)
	bit 5: reserved
	bit 6: reserved
	bit 7: force NVO update *)
	bInternalUseOnly : BYTE; (* Do not use this byte in your application! *)
END_STRUCT
END_TYPE

(* Data type in LON/NetworkVariables *)
TYPE typSnvtTimeStamp : 
STRUCT
	iYear : INT;
	bMonth : BYTE;
	bDay : BYTE;
	bHour : BYTE;
	bMinute : BYTE;
	bSecond : BYTE;
	bStatusInformation : BYTE; (* bit allocation of bStatusInformation:
	bit 0: NVI update counter LSB
	bit 1: NVI update counter
	bit 2: NVI update counter
	bit 3: NVI update counter MSB
	bit 4: timeout for NVI occurs (MaxRcvTime expired)
	bit 5: reserved
	bit 6: reserved
	bit 7: force NVO update *)
	bInternalUseOnly : BYTE; (* Do not use this byte in your application! *)
END_STRUCT
END_TYPE

(* POU PLC_PRG, ST *)
PROGRAM PLC_PRG
VAR
	Timer1: TON; (* Fast controls tick *)
	Timer2: TON; (* Plant control tick *)
	Timer3: TON; (* Logger timer *)

	T_CIR01		:	INT;
	T_CIR02		:	INT;
	T_CIR03		:	INT;
	T_CIRD01	:	INT;
	T_CIRD02	:	INT;

	T_Valve01	:	INT;
	T_Valve02	:	INT;
	T_Valve03	:	INT;
	T_Valve04	:	INT;
	T_Valve05	:	INT;

	SecCircuitLogic	:	BOOL;	(* Secondary circuit request: LOGICAL ON/OFF *)
	SecCircuitReal	:	BOOL;	(* Secondart circuit request: REAL ON/OFF	 *)

END_VAR
(******************************************************************************
 ****                           MAIN TASK CODE                             ****
 ******************************************************************************

	Network setup:
		IP  = 192.168.100.2 | MSK = 255.255.255.0
		GW	= 192.168.100.1 | DNS = 192.168.100.1
		SNTP = 193.204.114.232 (3600s) ==> 192.168.100.3

*)

(*==============================*)
(*===== Main status machine ====*)
(*==============================*)
Main_Stm();

(*==============================*)
(*== Running cycle operations ==*)
(*==============================*)
IF SYS.Status>S_INIT_VAR THEN
	(* Execute cycle processes *)
	(* Update LON output variables (needs to be here to obtain only one refresh) *)
	GRU01.Heartbeat( CLIM:=GRU01_Clima );
	(* Execute LON process *)
	Module_1_PRG();

	(* Count water pulses *)
	CTL01(CTL_ST:=CTL01_ST, COUNT:=Ctl01_Counter);
	CTL02(CTL_ST:=CTL02_ST, COUNT:=Ctl02_Counter);

	(* ModBus *)
	MODB01();

	CIR03(ModBus:=MODB01, Pump_AL:=NOT CIR03_AL, Pump_AUTO:=NOT CIR03_AUTO);

	CIRD01(ModBus:=MODB01, PumpA_AL:=NOT CIRD01_A_AL, PumpB_AL:=NOT CIRD01_B_AL, PumpA_AUTO:=NOT CIRD01_A_AUTO, PumpB_AUTO:=NOT CIRD01_B_AUTO);
	CIRD02(ModBus:=MODB01, PumpA_AL:=NOT CIRD02_A_AL, PumpB_AL:=NOT CIRD02_B_AL, PumpA_AUTO:=NOT CIRD02_A_AUTO, PumpB_AUTO:=NOT CIRD02_B_AUTO);

	(* TCP ModBus *)
	MODB02();

	ZTHL09(MODBUS:=MODB02);
	ZTHL10(MODBUS:=MODB02);
	ZTHL11(MODBUS:=MODB02);
	ZTHL12(MODBUS:=MODB02);
	ZTHL13(MODBUS:=MODB02);
	ZTHL14(MODBUS:=MODB02);

	(* M-Bus *)
	MBUS01();

	CTB01(MBUS:=MBUS01);
	CTB02(MBUS:=MBUS01);

END_IF

(*==============================*)
(*== System cycle operations ===*)
(*==============================*)
(* Execute TCP processes *)
Logger_Proc();
Remote_Proc();
(* Update user led *)
USRLED_Update();
(* Execute Cron Editor commands *)
CronEd();

(* Environment temperature *)
IF NOT TPV01.ERR THEN T_AMB := S01;
ELSE T_AMB := Plant_DefaultTAmb;
END_IF


(**** SIMULATION ONLY ****)
(*...*)
END_PROGRAM
ACTION Main_Stm:
CASE Sys.Status OF

	S_STARTUP:
		Sys.Status:=S_INIT_RTC;

	S_INIT_RTC:
		(* Check RTC and update from network *)
		RTC_Update();
		(* Check time *)
		IF Sys.Time_Year>2000 THEN
			Sys.Status:=S_INIT_VAR;
		END_IF

	S_INIT_VAR:
		LogEv(EL_Wrn,EO_SYS,0,1,CONCAT('System_startup_v',WORD_TO_STRING(Plant_SW_VER)));
		Sys.Status:=S_RUNNING;

	S_RUNNING:
		Timer1(IN:=NOT Timer1.Q,PT:=T#50ms);
		IF Timer1.Q THEN
			(* Update meters *)

			(* Update system checks *)
			SYS_Proc();
		END_IF

		Timer2(IN:=NOT Timer2.Q,PT:=T#500ms);
		IF Timer2.Q THEN
			(* Read current date/time *)
			RTC_Update();

			(* Secondary circuit heat request *)
			SecCircuitLogic := CIR01.Ctrl_Run AND CIR02.Ctrl_Run AND CIR03.Ctrl_Run AND CIRD01.Ctrl_Run AND CIRD02.Ctrl_Run;
			SecCircuitReal	:= CIR01.Run AND CIR02.Run AND CIR03.Run AND CIRD01.Run AND CIRD02.Run;

			GRU01.Run := SEL(SecCircuitLogic,FALSE,TRUE) AND SYS.AlarmStop=FALSE;

			GRU01(CLIM:=GRU01_Clima);

			(* Probes *)
			TPV01();
			TPV02();
			TPV03();
			TPV04();
			TPV05();
			TPV06();
			TPV07();
			TPV08();

			(* Temperature *)
			T_CIR01 := SEL(ZTHL11.fTemp,ZTHL11.OUT_TEMP,Plant_DefaultTAmb);
			T_CIR02 := SEL(ZTHL09.fTemp,ZTHL09.OUT_TEMP,Plant_DefaultTAmb);
			T_CIR03 := SEL(ZTHL12.fTemp,ZTHL12.OUT_TEMP,Plant_DefaultTAmb);
			T_CIRD01 := SEL(ZTHL10.fTemp,ZTHL10.OUT_TEMP,Plant_DefaultTAmb);

			T_CIRD02 := MUX_T(T1:=ZTHL13.OUT_TEMP, T2:=ZTHL14.OUT_TEMP, T3:=0,
							  Err1:=ZTHL13.fTemp, Err2:=ZTHL14.fTemp, Err3:=0, Used:=2);

			TPV04.Mean();
			T_Valve01 := SEL(TPV04.ERR,TPV04.AVG,Plant_VRD_TDefault);

			TPV05.Mean();
			T_Valve02 := SEL(TPV05.ERR,TPV05.AVG,Plant_VRD_TDefault);

			TPV06.Mean();
			T_Valve03 := SEL(TPV06.ERR,TPV06.AVG,Plant_VRD_TDefault);

			TPV07.Mean();
			T_Valve04 := SEL(TPV07.ERR,TPV07.AVG,Plant_VRD_TDefault);

			(* Thermostats *)
			THER01(Temperature:=T_CIR01, Run=>CIR01.OnOff, AntifreezeForce=>CIR01.CIR_RUN_REQ);
			THER02(Temperature:=T_CIR02, Run=>CIR02.OnOff, AntifreezeForce=>CIR02.CIR_RUN_REQ);
			THER03(Temperature:=T_CIR03, Run=>CIR03.OnOff, AntifreezeForce=>CIR03.CIR_RUN_REQ);
			THER04(Temperature:=T_CIRD01, Run=>CIRD01.OnOff, AntifreezeForce=>CIRD01.CIR_RUN_REQ);
			THER05(Temperature:=T_CIRD02, Run=>CIRD02.OnOff, AntifreezeForce=>CIRD02.CIR_RUN_REQ);

			(* CIR *)
			CIR01(Pump_AL:=NOT CIR01_AL, Pump_ST:=CIR01_ST, Pump_AUTO:=CIR01_AUTO);
			CIR02(Pump_AL:=NOT CIR02_AL, Pump_ST:=CIR02_ST, Pump_AUTO:=CIR02_AUTO);

			(* Valves *)
			VRD01(RUN:=CIRD02.Run, CLIM:=VRD01_Clima, TEMP:=T_Valve01, STATUS:=VRD01_ST, OUT_CL=>VRD01_CL, OUT_OP=>VRD01_OP);
			VRD02(RUN:=CIR03.Run, CLIM:=VRD02_Clima, TEMP:=T_Valve02, STATUS:=VRD02_ST, OUT_CL=>VRD02_CL, OUT_OP=>VRD02_OP);
			VRD03(RUN:=CIRD01.Run, CLIM:=VRD03_Clima, TEMP:=T_Valve03, STATUS:=VRD03_ST, OUT_CL=>VRD03_CL, OUT_OP=>VRD03_OP);
			VRD04(RUN:=CIR02.Run, CLIM:=VRD04_Clima, TEMP:=T_Valve04, STATUS:=VRD04_ST, OUT=>VRD04_CTRL);
			VRD05(RUN:=CIR01.Run, CLIM:=VRD05_Clima, TEMP:=T_Valve05, STATUS:=VRD05_ST, OUT=>VRD05_CTRL);


			(* Check plant status *)
			Lamp();

			(* Test toggle *)
			(*IF TEST1 THEN TEST1:=FALSE; ELSE TEST1:=TRUE; END_IF*)
		END_IF

		Timer3(IN:=NOT Timer3.Q,PT:=T#5m);
		IF Timer3.Q THEN
			(* Trig logger *)
			LogTrig();
			(* Execute temporary CSV logger *)
			(*CSV_Log();*)
		END_IF

	S_SHUTDOWN:
		(* Stop sistema *)
		Sys.Status:=S_STARTUP;

	S_HALT:
		(* Aspetta uscita manuale *)
		Sys.Status:=S_STARTUP;

ELSE
	Sys.Status:=S_STARTUP;
END_CASE;
END_ACTION

(* POU LON/Module_1/Module_1_PRG, FBD *)
PROGRAM Module_1_PRG
VAR
	(* Automatic added code, do not change! *)
	LonMaster : Module_1_LonMaster;
	SFPTnodeObject : Module_1_SFPTnodeObject;
	Virtualfunctionalblock : Module_1_Virtualfunctionalblock;

	InData_LON AT %IB24 : ARRAY[0..23] OF BYTE;
	OutData_LON AT %QB0 : ARRAY[0..23] OF BYTE;
	(***** End of automatic added code. *****)

	(* Add your code here. *)

	LonState: BOOL;
	LonReset: BOOL;
END_VAR
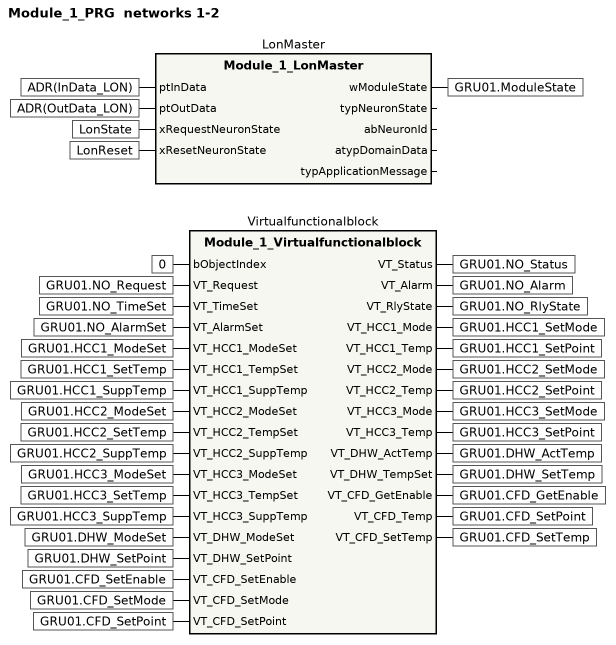
_FBD_ (* Function Block Diagram *)
NETWORK 1 (* Added by code generator *)
	LonMaster:Module_1_LonMaster(ptInData: ADR(InData_LON), ptOutData: ADR(OutData_LON), xRequestNeuronState: LonState, xResetNeuronState: LonReset) => GRU01.ModuleState
NETWORK 2
	Virtualfunctionalblock:Module_1_Virtualfunctionalblock(bObjectIndex: 0, VT_Request: GRU01.NO_Request, VT_TimeSet: GRU01.NO_TimeSet, VT_AlarmSet: GRU01.NO_AlarmSet, VT_HCC1_ModeSet: GRU01.HCC1_ModeSet, VT_HCC1_TempSet: GRU01.HCC1_SetTemp, VT_HCC1_SuppTemp: GRU01.HCC1_SuppTemp, VT_HCC2_ModeSet: GRU01.HCC2_ModeSet, VT_HCC2_TempSet: GRU01.HCC2_SetTemp, VT_HCC2_SuppTemp: GRU01.HCC2_SuppTemp, VT_HCC3_ModeSet: GRU01.HCC3_ModeSet, VT_HCC3_TempSet: GRU01.HCC3_SetTemp, VT_HCC3_SuppTemp: GRU01.HCC3_SuppTemp, VT_DHW_ModeSet: GRU01.DHW_ModeSet, VT_DHW_SetPoint: GRU01.DHW_SetPoint, VT_CFD_SetEnable: GRU01.CFD_SetEnable, VT_CFD_SetMode: GRU01.CFD_SetMode, VT_CFD_SetPoint: GRU01.CFD_SetPoint, VT_Alarm => GRU01.NO_Alarm, VT_RlyState => GRU01.NO_RlyState, VT_HCC1_Mode => GRU01.HCC1_SetMode, VT_HCC1_Temp => GRU01.HCC1_SetPoint, VT_HCC2_Mode => GRU01.HCC2_SetMode, VT_HCC2_Temp => GRU01.HCC2_SetPoint, VT_HCC3_Mode => GRU01.HCC3_SetMode, VT_HCC3_Temp => GRU01.HCC3_SetPoint, VT_DHW_ActTemp => GRU01.DHW_ActTemp, VT_DHW_TempSet => GRU01.DHW_SetTemp, VT_CFD_GetEnable => GRU01.CFD_GetEnable, VT_CFD_Temp => GRU01.CFD_SetPoint, VT_CFD_SetTemp => GRU01.CFD_SetTemp) => GRU01.NO_Status
_END_FBD_
(* the same logic as Structured Text *)
(* Network 1: Added by code generator *)
LonMaster(ptInData := ADR(InData_LON), ptOutData := ADR(OutData_LON), xRequestNeuronState := LonState, xResetNeuronState := LonReset);
GRU01.ModuleState := LonMaster.wModuleState;
(* Network 2 *)
Virtualfunctionalblock(bObjectIndex := 0, VT_Request := GRU01.NO_Request, VT_TimeSet := GRU01.NO_TimeSet, VT_AlarmSet := GRU01.NO_AlarmSet, VT_HCC1_ModeSet := GRU01.HCC1_ModeSet, VT_HCC1_TempSet := GRU01.HCC1_SetTemp, VT_HCC1_SuppTemp := GRU01.HCC1_SuppTemp, VT_HCC2_ModeSet := GRU01.HCC2_ModeSet, VT_HCC2_TempSet := GRU01.HCC2_SetTemp, VT_HCC2_SuppTemp := GRU01.HCC2_SuppTemp, VT_HCC3_ModeSet := GRU01.HCC3_ModeSet, VT_HCC3_TempSet := GRU01.HCC3_SetTemp, VT_HCC3_SuppTemp := GRU01.HCC3_SuppTemp, VT_DHW_ModeSet := GRU01.DHW_ModeSet, VT_DHW_SetPoint := GRU01.DHW_SetPoint, VT_CFD_SetEnable := GRU01.CFD_SetEnable, VT_CFD_SetMode := GRU01.CFD_SetMode, VT_CFD_SetPoint := GRU01.CFD_SetPoint);
GRU01.NO_Alarm := Virtualfunctionalblock.VT_Alarm;
GRU01.NO_RlyState := Virtualfunctionalblock.VT_RlyState;
GRU01.HCC1_SetMode := Virtualfunctionalblock.VT_HCC1_Mode;
GRU01.HCC1_SetPoint := Virtualfunctionalblock.VT_HCC1_Temp;
GRU01.HCC2_SetMode := Virtualfunctionalblock.VT_HCC2_Mode;
GRU01.HCC2_SetPoint := Virtualfunctionalblock.VT_HCC2_Temp;
GRU01.HCC3_SetMode := Virtualfunctionalblock.VT_HCC3_Mode;
GRU01.HCC3_SetPoint := Virtualfunctionalblock.VT_HCC3_Temp;
GRU01.DHW_ActTemp := Virtualfunctionalblock.VT_DHW_ActTemp;
GRU01.DHW_SetTemp := Virtualfunctionalblock.VT_DHW_TempSet;
GRU01.CFD_GetEnable := Virtualfunctionalblock.VT_CFD_GetEnable;
GRU01.CFD_SetPoint := Virtualfunctionalblock.VT_CFD_Temp;
GRU01.CFD_SetTemp := Virtualfunctionalblock.VT_CFD_SetTemp;
GRU01.NO_Status := Virtualfunctionalblock.VT_Status;
END_PROGRAM

(* POU LON/Module_1/Master/Module_1_LonMaster, ST *)
FUNCTION_BLOCK Module_1_LonMaster
(******************************************)
(* Automatic generated code, do not edit! *)
(******************************************)
VAR_INPUT
	ptInData  : POINTER TO BYTE;
	ptOutData : POINTER TO BYTE;
	xRequestNeuronState : BOOL;
	xResetNeuronState : BOOL;
END_VAR
VAR_OUTPUT
	wModuleState : WORD; (* bit coded wModuleState:
	15: communication to I/O-module interrupted (error)
	14 - 08: reserved
	07: ready for Neuron initialization
	06: Neuron active
	05: user interface active
	04: internal module communication interrupted (error)
	03: CP synchronization running
	02: Neuron is configured online
	01 - 00: reserved *)

	typNeuronState : NeuronState;
	abNeuronId : ARRAY[0..5] OF BYTE;
	atypDomainData : ARRAY[0..1] OF DomainData;
	typApplicationMessage : ApplicationMessageData;
END_VAR
VAR
	bInternalCode : BYTE;
	bNvIndex : BYTE;
	wCpIndex : WORD;
	lonCom : FbLonBasicCommunication;

	xInitIsStarted : BOOL := FALSE;

	TimeoutTimer : TON;
	timeOutTime : TIME := T#1000ms;
	xStateMachineIsChecked : BOOL;
	xTimerStart : BOOL;

	iDomainTable : INT;
	xSendRequestPending : BOOL;
	trigRequest : R_TRIG;
	trigReset : R_TRIG;

	abMbxRxPrio0Buf: ARRAY [0..309] OF BYTE;
	abMbxRxPrio1Buf: ARRAY [0..517] OF BYTE;
	aMbxRxBufSize: ARRAY [0..1] OF UINT := 310, 518;
	aMbxRxBufList: ARRAY [0..1] OF POINTER TO BYTE;
	afbMbxRxFb: ARRAY [0..1] OF MBX2_RX_DEFRAG;
	astMbxRxCtx: ARRAY [0..1] OF stMbx2DefragContext;

	abMbxTxPrio0Buf: ARRAY [0..309] OF BYTE;
	abMbxTxPrio1Buf: ARRAY [0..517] OF BYTE;
	aMbxTxBufSize: ARRAY [0..1] OF UINT := 310, 518;
	aMbxTxBufList: ARRAY [0..1] OF POINTER TO BYTE;
	afbMbxTxFb: ARRAY [0..1] OF MBX2_TX_FRAG;

	astMbxTrackContext: ARRAY [0..0] OF stMbx2TrackContext;
END_VAR
VAR CONSTANT
END_VAR
aMbxRxBufList[0] := ADR(abMbxRxPrio0Buf[0]);
aMbxRxBufList[1] := ADR(abMbxRxPrio1Buf[0]);

aMbxTxBufList[0] := ADR(abMbxTxPrio0Buf[0]);
aMbxTxBufList[1] := ADR(abMbxTxPrio1Buf[0]);

mbxModule_1.Ressources.pDefragBufList := ADR(aMbxRxBufList);
mbxModule_1.Ressources.pDefragBufSizeList := ADR(aMbxRxBufSize);
mbxModule_1.Ressources.pDefragCtxPtrList := ADR(astMbxRxCtx);
mbxModule_1.Ressources.pDefragFbList := ADR(afbMbxRxFb);
mbxModule_1.Ressources.pFragBufList := ADR(aMbxTxBufList);
mbxModule_1.Ressources.pFragBufSizeList := ADR(aMbxTxBufSize);
mbxModule_1.Ressources.pFragFbList := ADR(afbMbxTxFb);

mbxModule_1.Ressources.unMaxAvailableRxPrioIndex := 1;
mbxModule_1.Ressources.unMaxAvailableTxPrioIndex := 1;

mbxModule_1.Ressources.pTrackStList := ADR(astMbxTrackContext);
mbxModule_1.Ressources.unMaxAvailableTrackIndex := 0;

mbxModule_1.Ressources.pabRxWin := ptInData + 1;
mbxModule_1.Ressources.pabTxWin := ptOutData + 1;
mbxModule_1.Ressources.bTxWinSize := 23;
mbxModule_1.Ressources.bRxWinSize := 23;

IF (mbxModule_1.bStatus.2 = TRUE) OR (mbxModule_1.bStatus.1 = TRUE) THEN
	mbxModule_1.MBX_RESET();
	xInitRunning_Module_1 := TRUE;
	xInitIsStarted := FALSE;
END_IF
mbxModule_1.MBX_CYCLE();

IF (mbxModule_1.bStatus.0 <> TRUE) THEN 
	wModuleState := 16#8000;
	RETURN;
ELSE
	wModuleState.15 := FALSE;
END_IF

xStateMachineIsChecked := FALSE;
IF xInitRunning_Module_1 = TRUE THEN
	IF xInitIsStarted = FALSE THEN
		SetParameter();
		lonCom.eInitState := INIT_SND_SGNTR_REQ;
		lonCom.CheckInitState();
		xInitIsStarted := TRUE;
		xStateMachineIsChecked := TRUE;
	END_IF
END_IF

typApplicationMessage.xMsgRcvd := FALSE;
typApplicationMessage.xRspRcvd := FALSE;
ResetNviUpdate();
WHILE (mbxModule_1.xRxPending) DO
	unLastLen_mbxModule_1 := mbxModule_1.unRxLen;
	mbxModule_1.pbRxData := ADR(InDataTelegram_Module_1);
	mbxModule_1.MBX_RETRIEVE();
	IF (mbxModule_1.nError <> MBX_OK) THEN EXIT; END_IF;
	bInternalCode := InDataTelegram_Module_1[0];

	IF (xInitRunning_Module_1 = TRUE) AND (lonCom.eInitState <> INIT_TRANSFER_CFG) THEN
		IF (FuCheckForValidInitCode(bInternalCode)) THEN
			SetParameter();
			lonCom.unLastLen := unLastLen_mbxModule_1;
			lonCom.CheckInitState();
			xInitRunning_Module_1 := NOT lonCom.xInitDone;
			xStateMachineIsChecked := TRUE;
		END_IF
	END_IF

	IF (bInternalCode = M2C_NVI_UPDT_OCCD) OR (bInternalCode = M2C_NV_VALUE_RSP) OR (bInternalCode = M2C_NVI_UPDT_TOUT) THEN
		bNvIndex := InDataTelegram_Module_1[1];
		CASE bNvIndex OF
			0, 2, 4: Module_1_PRG.SFPTnodeObject.DataReceived();
			6, 8, 10, 12, 14, 17, 19, 22, 24, 27, 29, 31, 33, 35: Module_1_PRG.Virtualfunctionalblock.DataReceived();

		END_CASE;
	ELSIF (bInternalCode = M2C_CP_VALUE_RSP) THEN
		wCpIndex := InDataTelegram_Module_1[1] OR (InDataTelegram_Module_1[2] * 256);
		CASE wCpIndex OF

		END_CASE;
	ELSIF (bInternalCode = M2C_LON_MSG_RCVD) OR (bInternalCode = M2C_LON_RSP_RCVD) THEN
		ApplMsgReceived();
	ELSIF (bInternalCode = M2C_STATUS_RSP) THEN
		wModuleState := (wModuleState AND 16#FF00) + InDataTelegram_Module_1[1];
	ELSIF (bInternalCode = M2C_NEURON_ID) THEN
		FuMemCopy(ADR(InDataTelegram_Module_1[1]), ADR(abNeuronId), 6);
	ELSIF (bInternalCode = M2C_DOMAIN_DATA) THEN
		DomainDataRcvd();
	ELSIF (bInternalCode = M2C_MICRO_SERVER_STATUS_RSP) THEN
		NeuronStateRcvd();
	END_IF
END_WHILE

IF (xInitRunning_Module_1 = TRUE) AND ((lonCom.xCallStateMachine = TRUE) OR (TimeoutTimer.Q = TRUE)) AND (NOT xStateMachineIsChecked) THEN
	SetParameter();
	lonCom.xTimeOut := TimeoutTimer.Q;
	lonCom.CheckInitState();
END_IF
TimeoutTimer(IN:=lonCom.xTimerStart, PT:=timeOutTime);

trigRequest(CLK := xRequestNeuronState);
trigReset(CLK := xResetNeuronState);
IF (trigRequest.Q OR trigReset.Q) THEN
	RequestNeuronState();
END_IF
END_FUNCTION_BLOCK
ACTION ApplMsgReceived:
IF (InDataTelegram_Module_1[0] = M2C_LON_MSG_RCVD) THEN
	typApplicationMessage.typService := InDataTelegram_Module_1[1] AND 16#30;
	typApplicationMessage.bSourceSubnetId := InDataTelegram_Module_1[2];
	typApplicationMessage.bSourceNodeId := InDataTelegram_Module_1[3];
	typApplicationMessage.bCorrelator := InDataTelegram_Module_1[4];
	typApplicationMessage.bCode :=  InDataTelegram_Module_1[5];
	typApplicationMessage.bDataLength := UINT_TO_BYTE(unLastLen_mbxModule_1 - 6);
	IF typApplicationMessage.bDataLength > 48 THEN typApplicationMessage.bDataLength := 48; END_IF;
	FuMemSet(ADR(typApplicationMessage.abData), 0, SIZEOF(typApplicationMessage.abData));
	IF typApplicationMessage.bDataLength > 0 THEN
		FuMemCopy(ADR(InDataTelegram_Module_1[6]), ADR(typApplicationMessage.abData), typApplicationMessage.bDataLength);
	END_IF
	typApplicationMessage.xMsgRcvd := TRUE;
ELSE
	typApplicationMessage.typService := LON_RESPONSE;
	typApplicationMessage.bSourceSubnetId := InDataTelegram_Module_1[1];
	typApplicationMessage.bSourceNodeId := InDataTelegram_Module_1[2];
	typApplicationMessage.bCorrelator := 0;
	typApplicationMessage.bCode :=  InDataTelegram_Module_1[3];
	typApplicationMessage.bDataLength := UINT_TO_BYTE(unLastLen_mbxModule_1 - 4);
	IF typApplicationMessage.bDataLength > 48 THEN typApplicationMessage.bDataLength := 48; END_IF;
	FuMemSet(ADR(typApplicationMessage.abData), 0, SIZEOF(typApplicationMessage.abData));
	IF typApplicationMessage.bDataLength > 0 THEN
		FuMemCopy(ADR(InDataTelegram_Module_1[4]), ADR(typApplicationMessage.abData), typApplicationMessage.bDataLength);
	END_IF
	typApplicationMessage.xRspRcvd := TRUE;
END_IF
END_ACTION
ACTION DomainDataRcvd:
IF (unLastLen_mbxModule_1 = 17) THEN
	iDomainTable := InDataTelegram_Module_1[1];
	IF (iDomainTable < 0) OR (iDomainTable > 1) THEN RETURN; END_IF
	FuMemCopy(ADR(InDataTelegram_Module_1[2]), ADR(atypDomainData[iDomainTable].abDomainId), 6);
	atypDomainData[iDomainTable].bSubnet := InDataTelegram_Module_1[8];
	atypDomainData[iDomainTable].xIsNonClone := InDataTelegram_Module_1[9].7;
	atypDomainData[iDomainTable].bNodeId := InDataTelegram_Module_1[9] AND 16#7F;
	atypDomainData[iDomainTable].xIsInvalid := InDataTelegram_Module_1[10].7;
	atypDomainData[iDomainTable].bDomainIdLength := InDataTelegram_Module_1[10] AND 16#7F;
	FuMemCopy(ADR(InDataTelegram_Module_1[11]), ADR(atypDomainData[iDomainTable].abAuthenticationKey), 6);
END_IF
END_ACTION
ACTION NeuronStateRcvd:
IF (unLastLen_mbxModule_1 = 16) THEN
	typNeuronState.wCrcError := InDataTelegram_Module_1[1] + InDataTelegram_Module_1[2] * 256;
	typNeuronState.wTransactionTimeouts := InDataTelegram_Module_1[3] + InDataTelegram_Module_1[4] * 256;
	typNeuronState.wReceiveTransactionBuffersFull := InDataTelegram_Module_1[5] + InDataTelegram_Module_1[6] * 256;
	typNeuronState.wLostMessages := InDataTelegram_Module_1[7] + InDataTelegram_Module_1[8] * 256;
	typNeuronState.wMissedMessages := InDataTelegram_Module_1[9] + InDataTelegram_Module_1[10] * 256;
	typNeuronState.bResetCause := InDataTelegram_Module_1[11];
	typNeuronState.bNodeState := InDataTelegram_Module_1[12];
	typNeuronState.bFirmwareVersion := InDataTelegram_Module_1[13];
	typNeuronState.bLastErrorLogged := InDataTelegram_Module_1[14];
	typNeuronState.bModelNumber := InDataTelegram_Module_1[15];
END_IF
END_ACTION
ACTION RequestNeuronState:
OutDataTelegram_Module_1[0] := C2M_MICRO_SERVER_STATUS_QRY;
OutDataTelegram_Module_1[1] := BOOL_TO_BYTE(trigReset.Q);

mbxModule_1.bTxPrio := 1;
mbxModule_1.bTxProtID := 0;
mbxModule_1.pbTxData := ADR(OutDataTelegram_Module_1);
mbxModule_1.unTxLen := 2;
mbxModule_1.MBX_SEND();

IF (mbxModule_1.nError <> MBX_OK) THEN
	RETURN;
END_IF
END_ACTION
ACTION ResetNviUpdate:
Module_1_PRG.SFPTnodeObject.ResetNviUpdate();
Module_1_PRG.Virtualfunctionalblock.ResetNviUpdate();
END_ACTION
ACTION SetParameter:
lonCom.pMbx 			:= ADR(mbxModule_1);
lonCom.pInData 			:= ADR(InDataTelegram_Module_1);
lonCom.pOutData 		:= ADR(OutDataTelegram_Module_1);
lonCom.pTimer			:= ADR(TimeoutTimer);

lonCom.pActualSignature	:= ADR(abSignature_Module_1);
lonCom.pConfigBlock := ADR(abInterface_Module_1);
lonCom.wConfigSize 		:= wConfigSize_Module_1;
END_ACTION

(* POU LON/Module_1/NV_Interface/Module_1_SFPTnodeObject, ST *)
FUNCTION_BLOCK Module_1_SFPTnodeObject
(******************************************)
(* Automatic generated code, do not edit! *)
(******************************************)
VAR_INPUT
	bObjectIndex : BYTE := 0;
	nvoStatus : typSnvtObjStatus;
	nvoFileStat : typSnvtFileStatus;

END_VAR
VAR_OUTPUT
	nviRequest : typSnvtObjRequest;
	nviFileReq : typSnvtFileReq;
	nviFilePos : typSnvtFilePos;

END_VAR
VAR
	xSetOnce : BOOL := TRUE;
	xDataInUpdated : BOOL := FALSE;
	nvoStatusLast: typSnvtObjStatus;
	nvoFileStatLast: typSnvtFileStatus;

	cmd : BYTE;
	z : INT;
	bNvRelativeIdx : BYTE;
	bNvAbsoluteIdx : BYTE;
	wCpRelativeIdx : WORD;
	wCpAbsoluteIdx : WORD;
END_VAR
VAR CONSTANT
	bNvStartIndex : BYTE := 0;
	wCpStartIndex : WORD := 65535;
	bLmoCount : BYTE := 1;
END_VAR
IF (xInitRunning_Module_1 = TRUE) AND (xSetOnce = TRUE) THEN
	xSetOnce := FALSE;
	CachePointers();
	SetUpdateFlags();
END_IF

CheckUpdateFlags();
IF (xInitRunning_Module_1 = FALSE) AND (xDataInUpdated = FALSE) THEN
	IF (mbxModule_1.bStatus.0) THEN
		SendValueRequest();
	END_IF
END_IF

IF (xInitRunning_Module_1 = FALSE) AND (mbxModule_1.bStatus.0) THEN
	xSetOnce := TRUE;
	xDataInUpdated := FALSE;
	IF ((NOT FuMemCompare(ADR(nvoStatusLast), ADR(nvoStatus), ADR(nvoStatus.bStatusInformation) - ADR(nvoStatus))) OR (nvoStatus.bStatusInformation.7 = TRUE) OR (nvoStatusLast.bInternalUseOnly.1 = TRUE)) THEN
		FuSnvtObjStatusToRaw(ADR(nvoStatus), ADR(OutDataTelegram_Module_1[2]));

		bNvAbsoluteIdx := bNvStartIndex + bObjectIndex + (1 * bLmoCount);

		IF (FuDoNvoUpdate_Module_1(ADR(nvoStatus), ADR(nvoStatusLast), ADR(nvoStatus.bInternalUseOnly), ADR(nvoStatusLast.bInternalUseOnly), ADR(nvoStatus.bStatusInformation), bNvAbsoluteIdx, 6, SIZEOF(nvoStatus)) = FALSE) THEN
			RETURN;
		END_IF
	END_IF
	IF ((NOT FuMemCompare(ADR(nvoFileStatLast), ADR(nvoFileStat), ADR(nvoFileStat.bStatusInformation) - ADR(nvoFileStat))) OR (nvoFileStat.bStatusInformation.7 = TRUE) OR (nvoFileStatLast.bInternalUseOnly.1 = TRUE)) THEN
		FuSnvtFileStatusToRaw(ADR(nvoFileStat), ADR(OutDataTelegram_Module_1[2]));

		bNvAbsoluteIdx := bNvStartIndex + bObjectIndex + (3 * bLmoCount);

		IF (FuDoNvoUpdate_Module_1(ADR(nvoFileStat), ADR(nvoFileStatLast), ADR(nvoFileStat.bInternalUseOnly), ADR(nvoFileStatLast.bInternalUseOnly), ADR(nvoFileStat.bStatusInformation), bNvAbsoluteIdx, 27, SIZEOF(nvoFileStat)) = FALSE) THEN
			RETURN;
		END_IF
	END_IF

END_IF
END_FUNCTION_BLOCK
ACTION CachePointers:
;
END_ACTION
ACTION CheckUpdateFlags:
xDataInUpdated := (NOT nviRequest.bInternalUseOnly.0) AND (NOT nviFileReq.bInternalUseOnly.0) AND (NOT nviFilePos.bInternalUseOnly.0) AND TRUE;
END_ACTION
ACTION DataReceived:
cmd := InDataTelegram_Module_1[0];
IF (cmd = M2C_NVI_UPDT_OCCD) OR (cmd = M2C_NV_VALUE_RSP) OR (cmd = M2C_NVI_UPDT_TOUT) THEN
	bNvRelativeIdx := (InDataTelegram_Module_1[1] - bNvStartIndex - bObjectIndex) / bLmoCount;
	CASE bNvRelativeIdx OF
	0:
		IF (cmd = M2C_NVI_UPDT_OCCD) OR (cmd = M2C_NV_VALUE_RSP) THEN
			IF (unLastLen_mbxModule_1 = (2 + 3)) THEN
				FuRawToSnvtObjRequest(ADR(InDataTelegram_Module_1[2]), ADR(nviRequest));
				nviRequest.bInternalUseOnly.0 := FALSE;
				nviRequest.bStatusInformation := FuInkrementNviStatus(nviRequest.bStatusInformation);
			ELSIF (unLastLen_mbxModule_1 = 2) THEN
				nviRequest.bStatusInformation := FuInkrementNviStatus(nviRequest.bStatusInformation);
			END_IF
		ELSIF (cmd = M2C_NVI_UPDT_TOUT) THEN
			IF (unLastLen_mbxModule_1 = 3) THEN
				nviRequest.bStatusInformation.4 := BYTE_TO_BOOL(InDataTelegram_Module_1[2]);
			END_IF
		END_IF
	2:
		IF (cmd = M2C_NVI_UPDT_OCCD) OR (cmd = M2C_NV_VALUE_RSP) THEN
			IF (unLastLen_mbxModule_1 = (2 + 12)) THEN
				FuRawToSnvtFileReq(ADR(InDataTelegram_Module_1[2]), ADR(nviFileReq));
				nviFileReq.bInternalUseOnly.0 := FALSE;
				nviFileReq.bStatusInformation := FuInkrementNviStatus(nviFileReq.bStatusInformation);
			ELSIF (unLastLen_mbxModule_1 = 2) THEN
				nviFileReq.bStatusInformation := FuInkrementNviStatus(nviFileReq.bStatusInformation);
			END_IF
		ELSIF (cmd = M2C_NVI_UPDT_TOUT) THEN
			IF (unLastLen_mbxModule_1 = 3) THEN
				nviFileReq.bStatusInformation.4 := BYTE_TO_BOOL(InDataTelegram_Module_1[2]);
			END_IF
		END_IF
	4:
		IF (cmd = M2C_NVI_UPDT_OCCD) OR (cmd = M2C_NV_VALUE_RSP) THEN
			IF (unLastLen_mbxModule_1 = (2 + 6)) THEN
				FuRawToSnvtFilePos(ADR(InDataTelegram_Module_1[2]), ADR(nviFilePos));
				nviFilePos.bInternalUseOnly.0 := FALSE;
				nviFilePos.bStatusInformation := FuInkrementNviStatus(nviFilePos.bStatusInformation);
			ELSIF (unLastLen_mbxModule_1 = 2) THEN
				nviFilePos.bStatusInformation := FuInkrementNviStatus(nviFilePos.bStatusInformation);
			END_IF
		ELSIF (cmd = M2C_NVI_UPDT_TOUT) THEN
			IF (unLastLen_mbxModule_1 = 3) THEN
				nviFilePos.bStatusInformation.4 := BYTE_TO_BOOL(InDataTelegram_Module_1[2]);
			END_IF
		END_IF

	END_CASE
ELSIF (cmd = M2C_CP_VALUE_RSP) THEN
	wCpRelativeIdx := ((InDataTelegram_Module_1[1] + InDataTelegram_Module_1[2] * 256) - wCpStartIndex - bObjectIndex) / bLmoCount;
	CASE wCpRelativeIdx OF

	END_CASE
END_IF
END_ACTION
ACTION ResetNviUpdate:
nviRequest.bStatusInformation := nviRequest.bStatusInformation AND 16#F8;
nviFileReq.bStatusInformation := nviFileReq.bStatusInformation AND 16#F8;
nviFilePos.bStatusInformation := nviFilePos.bStatusInformation AND 16#F8;
;
END_ACTION
ACTION SendValueRequest:
IF (FuSendNviValueReq_Module_1(ADR(nviRequest.bInternalUseOnly), bNvStartIndex + bObjectIndex + (0 * bLmoCount)) = FALSE) THEN
	RETURN;
END_IF

IF (FuSendNviValueReq_Module_1(ADR(nviFileReq.bInternalUseOnly), bNvStartIndex + bObjectIndex + (2 * bLmoCount)) = FALSE) THEN
	RETURN;
END_IF

IF (FuSendNviValueReq_Module_1(ADR(nviFilePos.bInternalUseOnly), bNvStartIndex + bObjectIndex + (4 * bLmoCount)) = FALSE) THEN
	RETURN;
END_IF

;
END_ACTION
ACTION SetUpdateFlags:
nviRequest.bInternaluseOnly.0 := TRUE;
nvoStatusLast.bInternaluseOnly.1 := TRUE;
nvoStatusLast.bInternaluseOnly.7 := FALSE;
nviFileReq.bInternaluseOnly.0 := TRUE;
nvoFileStatLast.bInternaluseOnly.1 := TRUE;
nvoFileStatLast.bInternaluseOnly.7 := FALSE;
nviFilePos.bInternaluseOnly.0 := TRUE;
;
END_ACTION

(* POU LON/Shared/Internal/FuSnvtObjStatusToRaw, ST *)
FUNCTION FuSnvtObjStatusToRaw : BOOL
(******************************************)
(* Automatic generated code, do not edit! *)
(******************************************)
VAR_INPUT
	NvDataIn :  POINTER TO typSnvtObjStatus;
	DataOut : POINTER TO ARRAY[0..5] OF BYTE;
END_VAR
VAR
END_VAR
DataOut^[0] := WORD_TO_BYTE(SHR(NvDataIn^.wObjectId, 8));
DataOut^[1] := WORD_TO_BYTE(NvDataIn^.wObjectId);

DataOut^[2] := NvDataIn^.bBitfieldByteOffset2;

DataOut^[3] := NvDataIn^.bBitfieldByteOffset3;

DataOut^[4] := NvDataIn^.bBitfieldByteOffset4;

DataOut^[5] := NvDataIn^.bBitfieldByteOffset5;

FuSnvtObjStatusToRaw := TRUE;
END_FUNCTION

(* POU LON/Module_1/Internal/FuDoNvoUpdate_Module_1, ST *)
FUNCTION FuDoNvoUpdate_Module_1 : BOOL
(******************************************)
(* Automatic generated code, do not edit! *)
(******************************************)
VAR_INPUT
	ptNvo : POINTER TO BYTE;
	ptNvoLast : POINTER TO BYTE;
	ptNvoInternalUse : POINTER TO BYTE;
	ptNvoLastInternalUse : POINTER TO BYTE;
	ptNvoStatusInformation : POINTER TO BYTE;
	bNvoIndex : BYTE;
	uiNvoLength : UINT;
	uiNvoVariableLength : UINT;
END_VAR
IF (ptNvoLastInternalUse^.1 = TRUE) AND (ptNvoStatusInformation^.7 = FALSE) THEN
	OutDataTelegram_Module_1[0] := C2M_NV_VALUE;
ELSE
	OutDataTelegram_Module_1[0] := C2M_NVO_PROPAGATE;
END_IF
OutDataTelegram_Module_1[1] := bNvoIndex;

mbxModule_1.bTxPrio := BOOL_TO_BYTE(ptNvoLastInternalUse^.7);
mbxModule_1.bTxProtID := 0;
mbxModule_1.pbTxData := ADR(OutDataTelegram_Module_1);
mbxModule_1.unTxLen := 2 + uiNvoLength;
mbxModule_1.MBX_SEND();

IF (mbxModule_1.nError <> MBX_OK) THEN
	FuDoNvoUpdate_Module_1 := FALSE;
	RETURN;
END_IF

ptNvoLastInternalUse^.1 := FALSE;
ptNvoInternalUse^ := ptNvoLastInternalUse^;
FuMemCopy(ptNvo, ptNvoLast, uiNvoVariableLength);

FuDoNvoUpdate_Module_1 := TRUE;
END_FUNCTION

(* POU LON/Shared/Internal/FuSnvtFileStatusToRaw, ST *)
FUNCTION FuSnvtFileStatusToRaw : BOOL
(******************************************)
(* Automatic generated code, do not edit! *)
(******************************************)
VAR_INPUT
	NvDataIn :  POINTER TO typSnvtFileStatus;
	DataOut : POINTER TO ARRAY[0..26] OF BYTE;
END_VAR
VAR
END_VAR
DataOut^[0] := NvDataIn^.bStatus;

DataOut^[1] := WORD_TO_BYTE(SHR(NvDataIn^.wNumberOfFiles, 8));
DataOut^[2] := WORD_TO_BYTE(NvDataIn^.wNumberOfFiles);

DataOut^[3] := WORD_TO_BYTE(SHR(NvDataIn^.wSelectedFile, 8));
DataOut^[4] := WORD_TO_BYTE(NvDataIn^.wSelectedFile);

DataOut^[5] := NvDataIn^.abAdr[0];
DataOut^[6] := NvDataIn^.abAdr[1];
DataOut^[7] := NvDataIn^.abAdr[2];
DataOut^[8] := NvDataIn^.abAdr[3];
DataOut^[9] := NvDataIn^.abAdr[4];
DataOut^[10] := NvDataIn^.abAdr[5];
DataOut^[11] := NvDataIn^.abAdr[6];
DataOut^[12] := NvDataIn^.abAdr[7];
DataOut^[13] := NvDataIn^.abAdr[8];
DataOut^[14] := NvDataIn^.abAdr[9];
DataOut^[15] := NvDataIn^.abAdr[10];
DataOut^[16] := NvDataIn^.abAdr[11];
DataOut^[17] := NvDataIn^.abAdr[12];
DataOut^[18] := NvDataIn^.abAdr[13];
DataOut^[19] := NvDataIn^.abAdr[14];
DataOut^[20] := NvDataIn^.abAdr[15];
DataOut^[21] := NvDataIn^.abAdr[16];
DataOut^[22] := NvDataIn^.abAdr[17];
DataOut^[23] := NvDataIn^.abAdr[18];
DataOut^[24] := NvDataIn^.abAdr[19];
DataOut^[25] := NvDataIn^.abAdr[20];
DataOut^[26] := NvDataIn^.abAdr[21];

FuSnvtFileStatusToRaw := TRUE;
END_FUNCTION

(* POU LON/Module_1/Internal/FuSendNviValueReq_Module_1, ST *)
FUNCTION FuSendNviValueReq_Module_1 : BOOL
(******************************************)
(* Automatic generated code, do not edit! *)
(******************************************)
VAR_INPUT
	ptInternalUseOnly : POINTER TO BYTE;
	bNvIndex : BYTE;
END_VAR
IF ptInternalUseOnly^.0 = TRUE THEN
	OutDataTelegram_Module_1[0] := C2M_NV_VALUE_QRY;
	OutDataTelegram_Module_1[1] := bNvIndex;

	mbxModule_1.bTxPrio := 1;
	mbxModule_1.bTxProtID := 0;
	mbxModule_1.pbTxData := ADR(OutDataTelegram_Module_1);
	mbxModule_1.unTxLen := 2;
	mbxModule_1.MBX_SEND();

	IF (mbxModule_1.nError <> MBX_OK) THEN
		FuSendNviValueReq_Module_1 := FALSE;
		RETURN;
	END_IF
	ptInternalUseOnly^.0 := FALSE;
END_IF

FuSendNviValueReq_Module_1 := TRUE;
END_FUNCTION

(* POU LON/Module_1/NV_Interface/Module_1_Virtualfunctionalblock, ST *)
FUNCTION_BLOCK Module_1_Virtualfunctionalblock
(******************************************)
(* Automatic generated code, do not edit! *)
(******************************************)
VAR_INPUT
	bObjectIndex : BYTE := 0;
	VT_Request : typSnvtObjRequest;
	VT_TimeSet : typSnvtTimeStamp;
	VT_AlarmSet : typSnvtAlarm;
	VT_HCC1_ModeSet : typSnvtHvacMode;
	VT_HCC1_TempSet : typSnvtTempP;
	VT_HCC1_SuppTemp : typSnvtTempP;
	VT_HCC2_ModeSet : typSnvtHvacMode;
	VT_HCC2_TempSet : typSnvtTempP;
	VT_HCC2_SuppTemp : typSnvtTempP;
	VT_HCC3_ModeSet : typSnvtHvacMode;
	VT_HCC3_TempSet : typSnvtTempP;
	VT_HCC3_SuppTemp : typSnvtTempP;
	VT_DHW_ModeSet : typSnvtHvacMode;
	VT_DHW_SetPoint : typSnvtTempP;
	VT_CFD_SetEnable : typSnvtSwitch;
	VT_CFD_SetMode : typSnvtHvacMode;
	VT_CFD_SetPoint : typSnvtTempP;

END_VAR
VAR_OUTPUT
	VT_Status : typSnvtObjStatus;
	VT_Alarm : typSnvtAlarm;
	VT_RlyState : typSnvtState;
	VT_HCC1_Mode : typSnvtHvacMode;
	VT_HCC1_Temp : typSnvtTempP;
	VT_HCC2_Mode : typSnvtHvacMode;
	VT_HCC2_Temp : typSnvtTempP;
	VT_HCC3_Mode : typSnvtHvacMode;
	VT_HCC3_Temp : typSnvtTempP;
	VT_DHW_ActTemp : typSnvtTempP;
	VT_DHW_TempSet : typSnvtTempP;
	VT_CFD_GetEnable : typSnvtSwitch;
	VT_CFD_Temp : typSnvtTempP;
	VT_CFD_SetTemp : typSnvtTempP;

END_VAR
VAR
	xSetOnce : BOOL := TRUE;
	xDataInUpdated : BOOL := FALSE;
	VT_RequestLast: typSnvtObjRequest;
	VT_TimeSetLast: typSnvtTimeStamp;
	VT_AlarmSetLast: typSnvtAlarm;
	VT_CFD_SetEnableLast: typSnvtSwitch;
	paNviSnvtHvacMode : ARRAY[0..2] OF POINTER TO typSnvtHvacMode;
	aNviSnvtHvacModeIndex : ARRAY[0..2] OF BYTE := 7,12,17;
	paNviSnvtTempP : ARRAY[0..6] OF POINTER TO typSnvtTempP;
	aNviSnvtTempPIndex : ARRAY[0..6] OF BYTE := 9,14,19,22,24,28,30;
	paNvoSnvtHvacMode : ARRAY[0..4] OF POINTER TO typSnvtHvacMode;
	aNvoSnvtHvacModeIndex : ARRAY[0..4] OF BYTE := 6,11,16,21,27;
	aNvoSnvtHvacModeLast : ARRAY[0..4] OF typSnvtHvacMode;
	aNvoSnvtHvacModePriority : ARRAY[0..0] OF BYTE := 16#00;
	paNvoSnvtTempP : ARRAY[0..7] OF POINTER TO typSnvtTempP;
	aNvoSnvtTempPIndex : ARRAY[0..7] OF BYTE := 8,10,13,15,18,20,23,29;
	aNvoSnvtTempPLast : ARRAY[0..7] OF typSnvtTempP;
	aNvoSnvtTempPPriority : ARRAY[0..0] OF BYTE := 16#00;

	cmd : BYTE;
	z : INT;
	bNvRelativeIdx : BYTE;
	bNvAbsoluteIdx : BYTE;
	wCpRelativeIdx : WORD;
	wCpAbsoluteIdx : WORD;
END_VAR
VAR CONSTANT
	bNvStartIndex : BYTE := 5;
	wCpStartIndex : WORD := 65535;
	bLmoCount : BYTE := 1;
END_VAR
IF (xInitRunning_Module_1 = TRUE) AND (xSetOnce = TRUE) THEN
	xSetOnce := FALSE;
	CachePointers();
	SetUpdateFlags();
END_IF

CheckUpdateFlags();
IF (xInitRunning_Module_1 = FALSE) AND (xDataInUpdated = FALSE) THEN
	IF (mbxModule_1.bStatus.0) THEN
		SendValueRequest();
	END_IF
END_IF

IF (xInitRunning_Module_1 = FALSE) AND (mbxModule_1.bStatus.0) THEN
	xSetOnce := TRUE;
	xDataInUpdated := FALSE;
	IF ((NOT FuMemCompare(ADR(VT_RequestLast), ADR(VT_Request), ADR(VT_Request.bStatusInformation) - ADR(VT_Request))) OR (VT_Request.bStatusInformation.7 = TRUE) OR (VT_RequestLast.bInternalUseOnly.1 = TRUE)) THEN
		FuSnvtObjRequestToRaw(ADR(VT_Request), ADR(OutDataTelegram_Module_1[2]));

		bNvAbsoluteIdx := bNvStartIndex + bObjectIndex + (0 * bLmoCount);

		IF (FuDoNvoUpdate_Module_1(ADR(VT_Request), ADR(VT_RequestLast), ADR(VT_Request.bInternalUseOnly), ADR(VT_RequestLast.bInternalUseOnly), ADR(VT_Request.bStatusInformation), bNvAbsoluteIdx, 3, SIZEOF(VT_Request)) = FALSE) THEN
			RETURN;
		END_IF
	END_IF
	IF ((NOT FuMemCompare(ADR(VT_TimeSetLast), ADR(VT_TimeSet), ADR(VT_TimeSet.bStatusInformation) - ADR(VT_TimeSet))) OR (VT_TimeSet.bStatusInformation.7 = TRUE) OR (VT_TimeSetLast.bInternalUseOnly.1 = TRUE)) THEN
		FuSnvtTimeStampToRaw(ADR(VT_TimeSet), ADR(OutDataTelegram_Module_1[2]));

		bNvAbsoluteIdx := bNvStartIndex + bObjectIndex + (2 * bLmoCount);

		IF (FuDoNvoUpdate_Module_1(ADR(VT_TimeSet), ADR(VT_TimeSetLast), ADR(VT_TimeSet.bInternalUseOnly), ADR(VT_TimeSetLast.bInternalUseOnly), ADR(VT_TimeSet.bStatusInformation), bNvAbsoluteIdx, 7, SIZEOF(VT_TimeSet)) = FALSE) THEN
			RETURN;
		END_IF
	END_IF
	IF ((NOT FuMemCompare(ADR(VT_AlarmSetLast), ADR(VT_AlarmSet), ADR(VT_AlarmSet.bStatusInformation) - ADR(VT_AlarmSet))) OR (VT_AlarmSet.bStatusInformation.7 = TRUE) OR (VT_AlarmSetLast.bInternalUseOnly.1 = TRUE)) THEN
		FuSnvtAlarmToRaw(ADR(VT_AlarmSet), ADR(OutDataTelegram_Module_1[2]));

		bNvAbsoluteIdx := bNvStartIndex + bObjectIndex + (4 * bLmoCount);

		IF (FuDoNvoUpdate_Module_1(ADR(VT_AlarmSet), ADR(VT_AlarmSetLast), ADR(VT_AlarmSet.bInternalUseOnly), ADR(VT_AlarmSetLast.bInternalUseOnly), ADR(VT_AlarmSet.bStatusInformation), bNvAbsoluteIdx, 29, SIZEOF(VT_AlarmSet)) = FALSE) THEN
			RETURN;
		END_IF
	END_IF
	IF ((NOT FuMemCompare(ADR(VT_CFD_SetEnableLast), ADR(VT_CFD_SetEnable), ADR(VT_CFD_SetEnable.bStatusInformation) - ADR(VT_CFD_SetEnable))) OR (VT_CFD_SetEnable.bStatusInformation.7 = TRUE) OR (VT_CFD_SetEnableLast.bInternalUseOnly.1 = TRUE)) THEN
		FuSnvtSwitchToRaw(ADR(VT_CFD_SetEnable), ADR(OutDataTelegram_Module_1[2]));

		bNvAbsoluteIdx := bNvStartIndex + bObjectIndex + (25 * bLmoCount);

		IF (FuDoNvoUpdate_Module_1(ADR(VT_CFD_SetEnable), ADR(VT_CFD_SetEnableLast), ADR(VT_CFD_SetEnable.bInternalUseOnly), ADR(VT_CFD_SetEnableLast.bInternalUseOnly), ADR(VT_CFD_SetEnable.bStatusInformation), bNvAbsoluteIdx, 2, SIZEOF(VT_CFD_SetEnable)) = FALSE) THEN
			RETURN;
		END_IF
	END_IF
	FOR z := 0 TO 4 DO
		IF ((NOT FuMemCompare(ADR(aNvoSnvtHvacModeLast[z]), paNvoSnvtHvacMode[z], ADR(paNvoSnvtHvacMode[z]^.bStatusInformation) - paNvoSnvtHvacMode[z])) OR (paNvoSnvtHvacMode[z]^.bStatusInformation.7 = TRUE) OR (aNvoSnvtHvacModeLast[z].bInternalUseOnly.1 = TRUE)) THEN
			FuSnvtHvacModeToRaw(paNvoSnvtHvacMode[z], ADR(OutDataTelegram_Module_1[2]));

			bNvAbsoluteIdx := bNvStartIndex + bObjectIndex + (aNvoSnvtHvacModeIndex[z] * bLmoCount);

			IF (FuDoNvoUpdate_Module_1(paNvoSnvtHvacMode[z], ADR(aNvoSnvtHvacModeLast[z]), ADR(paNvoSnvtHvacMode[z]^.bInternalUseOnly), ADR(aNvoSnvtHvacModeLast[z].bInternalUseOnly), ADR(paNvoSnvtHvacMode[z]^.bStatusInformation), bNvAbsoluteIdx, 1, SIZEOF(aNvoSnvtHvacModeLast[z])) = FALSE) THEN
				RETURN;
			END_IF
		END_IF
	END_FOR
	FOR z := 0 TO 7 DO
		IF ((NOT FuMemCompare(ADR(aNvoSnvtTempPLast[z]), paNvoSnvtTempP[z], ADR(paNvoSnvtTempP[z]^.bStatusInformation) - paNvoSnvtTempP[z])) OR (paNvoSnvtTempP[z]^.bStatusInformation.7 = TRUE) OR (aNvoSnvtTempPLast[z].bInternalUseOnly.1 = TRUE)) THEN
			FuSnvtTempPToRaw(paNvoSnvtTempP[z], ADR(OutDataTelegram_Module_1[2]));

			bNvAbsoluteIdx := bNvStartIndex + bObjectIndex + (aNvoSnvtTempPIndex[z] * bLmoCount);

			IF (FuDoNvoUpdate_Module_1(paNvoSnvtTempP[z], ADR(aNvoSnvtTempPLast[z]), ADR(paNvoSnvtTempP[z]^.bInternalUseOnly), ADR(aNvoSnvtTempPLast[z].bInternalUseOnly), ADR(paNvoSnvtTempP[z]^.bStatusInformation), bNvAbsoluteIdx, 2, SIZEOF(aNvoSnvtTempPLast[z])) = FALSE) THEN
				RETURN;
			END_IF
		END_IF
	END_FOR

END_IF
END_FUNCTION_BLOCK
ACTION CachePointers:
paNviSnvtHvacMode[0] := ADR(VT_HCC1_Mode);
paNviSnvtHvacMode[1] := ADR(VT_HCC2_Mode);
paNviSnvtHvacMode[2] := ADR(VT_HCC3_Mode);
paNviSnvtTempP[0] := ADR(VT_HCC1_Temp);
paNviSnvtTempP[1] := ADR(VT_HCC2_Temp);
paNviSnvtTempP[2] := ADR(VT_HCC3_Temp);
paNviSnvtTempP[3] := ADR(VT_DHW_ActTemp);
paNviSnvtTempP[4] := ADR(VT_DHW_TempSet);
paNviSnvtTempP[5] := ADR(VT_CFD_Temp);
paNviSnvtTempP[6] := ADR(VT_CFD_SetTemp);
paNvoSnvtHvacMode[0] := ADR(VT_HCC1_ModeSet);
paNvoSnvtHvacMode[1] := ADR(VT_HCC2_ModeSet);
paNvoSnvtHvacMode[2] := ADR(VT_HCC3_ModeSet);
paNvoSnvtHvacMode[3] := ADR(VT_DHW_ModeSet);
paNvoSnvtHvacMode[4] := ADR(VT_CFD_SetMode);
paNvoSnvtTempP[0] := ADR(VT_HCC1_TempSet);
paNvoSnvtTempP[1] := ADR(VT_HCC1_SuppTemp);
paNvoSnvtTempP[2] := ADR(VT_HCC2_TempSet);
paNvoSnvtTempP[3] := ADR(VT_HCC2_SuppTemp);
paNvoSnvtTempP[4] := ADR(VT_HCC3_TempSet);
paNvoSnvtTempP[5] := ADR(VT_HCC3_SuppTemp);
paNvoSnvtTempP[6] := ADR(VT_DHW_SetPoint);
paNvoSnvtTempP[7] := ADR(VT_CFD_SetPoint);
;
END_ACTION
ACTION CheckUpdateFlags:
xDataInUpdated := (NOT VT_Status.bInternalUseOnly.0) AND (NOT VT_Alarm.bInternalUseOnly.0) AND (NOT VT_RlyState.bInternalUseOnly.0) AND (NOT VT_CFD_GetEnable.bInternalUseOnly.0) AND TRUE;
FOR z := 0 TO 2 DO
	xDataInUpdated := xDataInUpdated AND (NOT paNviSnvtHvacMode[z]^.bInternalUseOnly.0);
END_FOR
FOR z := 0 TO 6 DO
	xDataInUpdated := xDataInUpdated AND (NOT paNviSnvtTempP[z]^.bInternalUseOnly.0);
END_FOR
END_ACTION
ACTION DataReceived:
cmd := InDataTelegram_Module_1[0];
IF (cmd = M2C_NVI_UPDT_OCCD) OR (cmd = M2C_NV_VALUE_RSP) OR (cmd = M2C_NVI_UPDT_TOUT) THEN
	bNvRelativeIdx := (InDataTelegram_Module_1[1] - bNvStartIndex - bObjectIndex) / bLmoCount;
	CASE bNvRelativeIdx OF
	1:
		IF (cmd = M2C_NVI_UPDT_OCCD) OR (cmd = M2C_NV_VALUE_RSP) THEN
			IF (unLastLen_mbxModule_1 = (2 + 6)) THEN
				FuRawToSnvtObjStatus(ADR(InDataTelegram_Module_1[2]), ADR(VT_Status));
				VT_Status.bInternalUseOnly.0 := FALSE;
				VT_Status.bStatusInformation := FuInkrementNviStatus(VT_Status.bStatusInformation);
			ELSIF (unLastLen_mbxModule_1 = 2) THEN
				VT_Status.bStatusInformation := FuInkrementNviStatus(VT_Status.bStatusInformation);
			END_IF
		ELSIF (cmd = M2C_NVI_UPDT_TOUT) THEN
			IF (unLastLen_mbxModule_1 = 3) THEN
				VT_Status.bStatusInformation.4 := BYTE_TO_BOOL(InDataTelegram_Module_1[2]);
			END_IF
		END_IF
	3:
		IF (cmd = M2C_NVI_UPDT_OCCD) OR (cmd = M2C_NV_VALUE_RSP) THEN
			IF (unLastLen_mbxModule_1 = (2 + 29)) THEN
				FuRawToSnvtAlarm(ADR(InDataTelegram_Module_1[2]), ADR(VT_Alarm));
				VT_Alarm.bInternalUseOnly.0 := FALSE;
				VT_Alarm.bStatusInformation := FuInkrementNviStatus(VT_Alarm.bStatusInformation);
			ELSIF (unLastLen_mbxModule_1 = 2) THEN
				VT_Alarm.bStatusInformation := FuInkrementNviStatus(VT_Alarm.bStatusInformation);
			END_IF
		ELSIF (cmd = M2C_NVI_UPDT_TOUT) THEN
			IF (unLastLen_mbxModule_1 = 3) THEN
				VT_Alarm.bStatusInformation.4 := BYTE_TO_BOOL(InDataTelegram_Module_1[2]);
			END_IF
		END_IF
	5:
		IF (cmd = M2C_NVI_UPDT_OCCD) OR (cmd = M2C_NV_VALUE_RSP) THEN
			IF (unLastLen_mbxModule_1 = (2 + 2)) THEN
				FuRawToSnvtState(ADR(InDataTelegram_Module_1[2]), ADR(VT_RlyState));
				VT_RlyState.bInternalUseOnly.0 := FALSE;
				VT_RlyState.bStatusInformation := FuInkrementNviStatus(VT_RlyState.bStatusInformation);
			ELSIF (unLastLen_mbxModule_1 = 2) THEN
				VT_RlyState.bStatusInformation := FuInkrementNviStatus(VT_RlyState.bStatusInformation);
			END_IF
		ELSIF (cmd = M2C_NVI_UPDT_TOUT) THEN
			IF (unLastLen_mbxModule_1 = 3) THEN
				VT_RlyState.bStatusInformation.4 := BYTE_TO_BOOL(InDataTelegram_Module_1[2]);
			END_IF
		END_IF
	26:
		IF (cmd = M2C_NVI_UPDT_OCCD) OR (cmd = M2C_NV_VALUE_RSP) THEN
			IF (unLastLen_mbxModule_1 = (2 + 2)) THEN
				FuRawToSnvtSwitch(ADR(InDataTelegram_Module_1[2]), ADR(VT_CFD_GetEnable));
				VT_CFD_GetEnable.bInternalUseOnly.0 := FALSE;
				VT_CFD_GetEnable.bStatusInformation := FuInkrementNviStatus(VT_CFD_GetEnable.bStatusInformation);
			ELSIF (unLastLen_mbxModule_1 = 2) THEN
				VT_CFD_GetEnable.bStatusInformation := FuInkrementNviStatus(VT_CFD_GetEnable.bStatusInformation);
			END_IF
		ELSIF (cmd = M2C_NVI_UPDT_TOUT) THEN
			IF (unLastLen_mbxModule_1 = 3) THEN
				VT_CFD_GetEnable.bStatusInformation.4 := BYTE_TO_BOOL(InDataTelegram_Module_1[2]);
			END_IF
		END_IF
	7, 12, 17:
		IF (cmd = M2C_NVI_UPDT_OCCD) OR (cmd = M2C_NV_VALUE_RSP) THEN
			IF (unLastLen_mbxModule_1 = (2 + 1)) THEN
				FOR z := 0 TO 2 DO
					IF aNviSnvtHvacModeIndex[z] = bNvRelativeIdx THEN
						FuRawToSnvtHvacMode(ADR(InDataTelegram_Module_1[2]), paNviSnvtHvacMode[z]);
						paNviSnvtHvacMode[z]^.bInternalUseOnly.0 := FALSE;
						paNviSnvtHvacMode[z]^.bStatusInformation := FuInkrementNviStatus(paNviSnvtHvacMode[z]^.bStatusInformation);
						EXIT;
					END_IF
				END_FOR
			ELSIF (unLastLen_mbxModule_1 = 2) THEN
				FOR z := 0 TO 2 DO
					IF aNviSnvtHvacModeIndex[z] = bNvRelativeIdx THEN
						paNviSnvtHvacMode[z]^.bStatusInformation := FuInkrementNviStatus(paNviSnvtHvacMode[z]^.bStatusInformation);
						EXIT;
					END_IF
				END_FOR
			END_IF
		ELSIF (cmd = M2C_NVI_UPDT_TOUT) THEN
			IF (unLastLen_mbxModule_1 = 3) THEN
				FOR z := 0 TO 2 DO
					IF aNviSnvtHvacModeIndex[z] = bNvRelativeIdx THEN
						paNviSnvtHvacMode[z]^.bStatusInformation.4 := BYTE_TO_BOOL(InDataTelegram_Module_1[2]);
						EXIT;
					END_IF
				END_FOR
			END_IF
		END_IF
	9, 14, 19, 22, 24, 28, 30:
		IF (cmd = M2C_NVI_UPDT_OCCD) OR (cmd = M2C_NV_VALUE_RSP) THEN
			IF (unLastLen_mbxModule_1 = (2 + 2)) THEN
				FOR z := 0 TO 6 DO
					IF aNviSnvtTempPIndex[z] = bNvRelativeIdx THEN
						FuRawToSnvtTempP(ADR(InDataTelegram_Module_1[2]), paNviSnvtTempP[z]);
						paNviSnvtTempP[z]^.bInternalUseOnly.0 := FALSE;
						paNviSnvtTempP[z]^.bStatusInformation := FuInkrementNviStatus(paNviSnvtTempP[z]^.bStatusInformation);
						EXIT;
					END_IF
				END_FOR
			ELSIF (unLastLen_mbxModule_1 = 2) THEN
				FOR z := 0 TO 6 DO
					IF aNviSnvtTempPIndex[z] = bNvRelativeIdx THEN
						paNviSnvtTempP[z]^.bStatusInformation := FuInkrementNviStatus(paNviSnvtTempP[z]^.bStatusInformation);
						EXIT;
					END_IF
				END_FOR
			END_IF
		ELSIF (cmd = M2C_NVI_UPDT_TOUT) THEN
			IF (unLastLen_mbxModule_1 = 3) THEN
				FOR z := 0 TO 6 DO
					IF aNviSnvtTempPIndex[z] = bNvRelativeIdx THEN
						paNviSnvtTempP[z]^.bStatusInformation.4 := BYTE_TO_BOOL(InDataTelegram_Module_1[2]);
						EXIT;
					END_IF
				END_FOR
			END_IF
		END_IF

	END_CASE
ELSIF (cmd = M2C_CP_VALUE_RSP) THEN
	wCpRelativeIdx := ((InDataTelegram_Module_1[1] + InDataTelegram_Module_1[2] * 256) - wCpStartIndex - bObjectIndex) / bLmoCount;
	CASE wCpRelativeIdx OF

	END_CASE
END_IF
END_ACTION
ACTION ResetNviUpdate:
VT_Status.bStatusInformation := VT_Status.bStatusInformation AND 16#F8;
VT_Alarm.bStatusInformation := VT_Alarm.bStatusInformation AND 16#F8;
VT_RlyState.bStatusInformation := VT_RlyState.bStatusInformation AND 16#F8;
VT_CFD_GetEnable.bStatusInformation := VT_CFD_GetEnable.bStatusInformation AND 16#F8;
FOR z := 0 TO 2 DO
	paNviSnvtHvacMode[z]^.bStatusInformation := paNviSnvtHvacMode[z]^.bStatusInformation AND 16#F8;
END_FOR
FOR z := 0 TO 6 DO
	paNviSnvtTempP[z]^.bStatusInformation := paNviSnvtTempP[z]^.bStatusInformation AND 16#F8;
END_FOR
;
END_ACTION
ACTION SendValueRequest:
IF (FuSendNviValueReq_Module_1(ADR(VT_Status.bInternalUseOnly), bNvStartIndex + bObjectIndex + (1 * bLmoCount)) = FALSE) THEN
	RETURN;
END_IF

IF (FuSendNviValueReq_Module_1(ADR(VT_Alarm.bInternalUseOnly), bNvStartIndex + bObjectIndex + (3 * bLmoCount)) = FALSE) THEN
	RETURN;
END_IF

IF (FuSendNviValueReq_Module_1(ADR(VT_RlyState.bInternalUseOnly), bNvStartIndex + bObjectIndex + (5 * bLmoCount)) = FALSE) THEN
	RETURN;
END_IF

IF (FuSendNviValueReq_Module_1(ADR(VT_CFD_GetEnable.bInternalUseOnly), bNvStartIndex + bObjectIndex + (26 * bLmoCount)) = FALSE) THEN
	RETURN;
END_IF

FOR z := 0 TO 2 DO
	IF (FuSendNviValueReq_Module_1(ADR(paNviSnvtHvacMode[z]^.bInternalUseOnly), bNvStartIndex + bObjectIndex + (aNviSnvtHvacModeIndex[z] * bLmoCount)) = FALSE) THEN
		RETURN;
	END_IF;
END_FOR;
FOR z := 0 TO 6 DO
	IF (FuSendNviValueReq_Module_1(ADR(paNviSnvtTempP[z]^.bInternalUseOnly), bNvStartIndex + bObjectIndex + (aNviSnvtTempPIndex[z] * bLmoCount)) = FALSE) THEN
		RETURN;
	END_IF;
END_FOR;
;
END_ACTION
ACTION SetUpdateFlags:
VT_RequestLast.bInternaluseOnly.1 := TRUE;
VT_RequestLast.bInternaluseOnly.7 := FALSE;
VT_Status.bInternaluseOnly.0 := TRUE;
VT_TimeSetLast.bInternaluseOnly.1 := TRUE;
VT_TimeSetLast.bInternaluseOnly.7 := FALSE;
VT_Alarm.bInternaluseOnly.0 := TRUE;
VT_AlarmSetLast.bInternaluseOnly.1 := TRUE;
VT_AlarmSetLast.bInternaluseOnly.7 := FALSE;
VT_RlyState.bInternaluseOnly.0 := TRUE;
VT_CFD_SetEnableLast.bInternaluseOnly.1 := TRUE;
VT_CFD_SetEnableLast.bInternaluseOnly.7 := FALSE;
VT_CFD_GetEnable.bInternaluseOnly.0 := TRUE;
FOR z := 0 TO 2 DO
	paNviSnvtHvacMode[z]^.bInternaluseOnly.0 := TRUE;
END_FOR;
FOR z := 0 TO 6 DO
	paNviSnvtTempP[z]^.bInternaluseOnly.0 := TRUE;
END_FOR;
FOR z := 0 TO 4 DO
	aNvoSnvtHvacModeLast[z].bInternaluseOnly.1 := TRUE;
	aNvoSnvtHvacModeLast[z].bInternaluseOnly.7 := (SHR(aNvoSnvtHvacModePriority[z / 8], z MOD 8) AND 1) <> 0;
END_FOR;
FOR z := 0 TO 7 DO
	aNvoSnvtTempPLast[z].bInternaluseOnly.1 := TRUE;
	aNvoSnvtTempPLast[z].bInternaluseOnly.7 := (SHR(aNvoSnvtTempPPriority[z / 8], z MOD 8) AND 1) <> 0;
END_FOR;
;
END_ACTION

(* POU LON/Shared/Internal/FuSnvtObjRequestToRaw, ST *)
FUNCTION FuSnvtObjRequestToRaw : BOOL
(******************************************)
(* Automatic generated code, do not edit! *)
(******************************************)
VAR_INPUT
	NvDataIn :  POINTER TO typSnvtObjRequest;
	DataOut : POINTER TO ARRAY[0..2] OF BYTE;
END_VAR
VAR
END_VAR
DataOut^[0] := WORD_TO_BYTE(SHR(NvDataIn^.wObjectId, 8));
DataOut^[1] := WORD_TO_BYTE(NvDataIn^.wObjectId);

DataOut^[2] := NvDataIn^.bObjectRequest;

FuSnvtObjRequestToRaw := TRUE;
END_FUNCTION

(* POU LON/Shared/Internal/FuSnvtTimeStampToRaw, ST *)
FUNCTION FuSnvtTimeStampToRaw : BOOL
(******************************************)
(* Automatic generated code, do not edit! *)
(******************************************)
VAR_INPUT
	NvDataIn :  POINTER TO typSnvtTimeStamp;
	DataOut : POINTER TO ARRAY[0..6] OF BYTE;
END_VAR
VAR
END_VAR
DataOut^[0] := INT_TO_BYTE(SHR(NvDataIn^.iYear, 8));
DataOut^[1] := INT_TO_BYTE(NvDataIn^.iYear);

DataOut^[2] := NvDataIn^.bMonth;

DataOut^[3] := NvDataIn^.bDay;

DataOut^[4] := NvDataIn^.bHour;

DataOut^[5] := NvDataIn^.bMinute;

DataOut^[6] := NvDataIn^.bSecond;

FuSnvtTimeStampToRaw := TRUE;
END_FUNCTION

(* POU LON/Shared/Internal/FuSnvtAlarmToRaw, ST *)
FUNCTION FuSnvtAlarmToRaw : BOOL
(******************************************)
(* Automatic generated code, do not edit! *)
(******************************************)
VAR_INPUT
	NvDataIn :  POINTER TO typSnvtAlarm;
	DataOut : POINTER TO ARRAY[0..28] OF BYTE;
END_VAR
VAR
END_VAR
DataOut^[0] := NvDataIn^.abLocation[0];
DataOut^[1] := NvDataIn^.abLocation[1];
DataOut^[2] := NvDataIn^.abLocation[2];
DataOut^[3] := NvDataIn^.abLocation[3];
DataOut^[4] := NvDataIn^.abLocation[4];
DataOut^[5] := NvDataIn^.abLocation[5];

DataOut^[6] := WORD_TO_BYTE(SHR(NvDataIn^.wObjectId, 8));
DataOut^[7] := WORD_TO_BYTE(NvDataIn^.wObjectId);

DataOut^[8] := NvDataIn^.bAlarmType;

DataOut^[9] := NvDataIn^.bPriorityLevel;

DataOut^[10] := WORD_TO_BYTE(SHR(NvDataIn^.wIndexToSnvt, 8));
DataOut^[11] := WORD_TO_BYTE(NvDataIn^.wIndexToSnvt);

DataOut^[12] := NvDataIn^.abValue[0];
DataOut^[13] := NvDataIn^.abValue[1];
DataOut^[14] := NvDataIn^.abValue[2];
DataOut^[15] := NvDataIn^.abValue[3];

DataOut^[16] := WORD_TO_BYTE(SHR(NvDataIn^.wYear, 8));
DataOut^[17] := WORD_TO_BYTE(NvDataIn^.wYear);

DataOut^[18] := NvDataIn^.bMonth;

DataOut^[19] := NvDataIn^.bDay;

DataOut^[20] := NvDataIn^.bHour;

DataOut^[21] := NvDataIn^.bMinute;

DataOut^[22] := NvDataIn^.bSecond;

DataOut^[23] := WORD_TO_BYTE(SHR(NvDataIn^.wMillisecond, 8));
DataOut^[24] := WORD_TO_BYTE(NvDataIn^.wMillisecond);

DataOut^[25] := NvDataIn^.abAlarmLimit[0];
DataOut^[26] := NvDataIn^.abAlarmLimit[1];
DataOut^[27] := NvDataIn^.abAlarmLimit[2];
DataOut^[28] := NvDataIn^.abAlarmLimit[3];

FuSnvtAlarmToRaw := TRUE;
END_FUNCTION

(* POU LON/Shared/Internal/FuSnvtSwitchToRaw, ST *)
FUNCTION FuSnvtSwitchToRaw : BOOL
(******************************************)
(* Automatic generated code, do not edit! *)
(******************************************)
VAR_INPUT
	NvDataIn :  POINTER TO typSnvtSwitch;
	DataOut : POINTER TO ARRAY[0..1] OF BYTE;
END_VAR
VAR
END_VAR
DataOut^[0] := NvDataIn^.bValue;

DataOut^[1] := NvDataIn^.siState;

FuSnvtSwitchToRaw := TRUE;
END_FUNCTION

(* POU LON/Shared/Internal/FuSnvtHvacModeToRaw, ST *)
FUNCTION FuSnvtHvacModeToRaw : BOOL
(******************************************)
(* Automatic generated code, do not edit! *)
(******************************************)
VAR_INPUT
	NvDataIn :  POINTER TO typSnvtHvacMode;
	DataOut : POINTER TO ARRAY[0..0] OF BYTE;
END_VAR
VAR
END_VAR
DataOut^[0] := NvDataIn^.bSnvtHvacMode;

FuSnvtHvacModeToRaw := TRUE;
END_FUNCTION

(* POU LON/Shared/Internal/FuSnvtTempPToRaw, ST *)
FUNCTION FuSnvtTempPToRaw : BOOL
(******************************************)
(* Automatic generated code, do not edit! *)
(******************************************)
VAR_INPUT
	NvDataIn :  POINTER TO typSnvtTempP;
	DataOut : POINTER TO ARRAY[0..1] OF BYTE;
END_VAR
VAR
END_VAR
DataOut^[0] := INT_TO_BYTE(SHR(NvDataIn^.iSnvtTempP, 8));
DataOut^[1] := INT_TO_BYTE(NvDataIn^.iSnvtTempP);

FuSnvtTempPToRaw := TRUE;
END_FUNCTION

(* POU TCP_Logger/Logger_Proc, ST *)
PROGRAM Logger_Proc
VAR
	c1:         	TCPCLIENT;

	Open:	    	BOOL;
	IpAddr:			DWORD;
	InetAddr:		DWORD;
	Connected:  	BOOL;
	Error:      	DINT;
	TxTrig:     	BOOL;
	RxData:			ARRAY [0..MAX_RECEIVE_TCP_CLIENT] OF BYTE;
	RxLen:			DINT;

	Retry:			BYTE;	(* Counter for connection retries *)
	Recovered:		BYTE;	(* Counter for recovered unsent messages *)

	i:				DINT;
	pos:			DWORD;
	hFile:			DWORD;

END_VAR
(*=== State machine ===*)
CASE Logger.Status OF

	S_Logger_UNKNOWN:
		(* Startup *)
		Logger.SendReq:=FALSE;
		Open:=FALSE;
		Logger.Status:=S_Logger_IDLE;

	S_Logger_IDLE:
		(* Wait request *)
		IF Logger.SendReq THEN
			(* Resolve server name or use static IP *)
			IF LEN(Logger_SERVER)=0 THEN
				InetAddr:=SysSockInetAddr(Logger_IP);
			ELSE
				IpAddr:=SysSockGetHostByName(ADR(Logger_SERVER));
				DWORDSWAP(pIn:=ADR(IpAddr), pOut:=ADR(InetAddr));
			END_IF
			TxTrig:=FALSE;
			RxLen:=0;
			(* Open connection *)
			Open:=TRUE;
			Logger.Status:=S_Logger_WAITCONN;
		END_IF

	S_Logger_WAITCONN:
		(* Wait connection *)
		IF Connected THEN
			(* Send data *)
			TxTrig:=TRUE;
			Logger.Status:=S_Logger_WAITTX;
		END_IF
		IF Error>0 THEN
			Open:=FALSE;
			Logger.Status:=S_Logger_ERROR;
		END_IF

	S_Logger_WAITTX:
		(* Wait transmission *)
		IF NOT TxTrig THEN
			Logger.Status:=S_Logger_WAITRESP;
		END_IF
		IF Error>0 THEN
			Open:=FALSE;
			Logger.Status:=S_Logger_ERROR;
		END_IF

	S_Logger_WAITRESP:
		(* Wait response *)
		IF Connected=FALSE (* OR TIMEOUT!! *) THEN
			Open:=FALSE;
			(* Check response *)
			IF RxLen>=4 AND CHKSTRING(pString:=ADR(RxData), pPattern:=ADR(Logger_CHECK)) THEN
				Logger.SendReq:=FALSE;
				Retry:=0;
				(* Check unsent messages to flush *)
				IF Recovered<Logger_RecoverMsgs THEN
					MsgChk();
					IF Logger.SendReq=TRUE THEN
						Recovered:=Recovered+1;
					ELSE
						Recovered:=0;
					END_IF
				ELSE
					Recovered:=0;
				END_IF
				Logger.Status:=S_Logger_IDLE;
			ELSE
				Logger.Status:=S_Logger_ERROR;
			END_IF
		END_IF

	S_Logger_ERROR:
		(* Connection error or send failure *)
		Retry:=Retry+1;
		IF Retry>Logger_ConnRetries THEN
			(* Save message as unsent *)
			MsgSave();
			Logger.SendReq:=FALSE;
			Retry:=0;
		END_IF
		Logger.Status:=S_Logger_IDLE;

ELSE
	Logger.Status:=S_Logger_UNKNOWN;
END_CASE


(*=== Execute client lib ===*)
c1(
	xOpenConnection			:= Open,
	dwInetAddr 				:= InetAddr,
	wPortNumber				:= Logger_PORT,
	ptSendData				:= ADR(Logger.SendData),
	diSendCount				:= Logger.SendLen,
	tConnectWatchdogTime	:= t#10s,
	xStartSend				:= TxTrig,
	aReceiveBuffer			:= RxData,
	diReceiveCount			:= RxLen,
	xConnected				=> Connected,
	diError					=> Error
);

(*=== Process Rx data ===*)
(*IF RxLen>0 THEN
	RxLen:=0;
END_IF*)
END_PROGRAM
ACTION MsgChk:
(* Open index file *)
hFile:=SysFileOpen(Logger_IndexFile,'r');
IF hFile=0 THEN
	RETURN;
END_IF
(* Search oldest message to recover *)
SysFileSetPos(hFile,Logger.LastIdxPos);
Logger.SendLen:=0;
REPEAT
	SysFileRead(hFile, ADR(Logger.SendIdx), SIZEOF(Logger.SendIdx));
	pos:=SysFileGetPos(hFile);
	SysFileRead(hFile, ADR(Logger.SendLen), SIZEOF(Logger.SendLen));
UNTIL
	SysFileEOF(hFile) OR Logger.SendLen<>0
END_REPEAT
SysFileClose(hFile);
(* Delete index file when all messages are recovered *)
IF Logger.SendLen=0 THEN
	Logger.LastIdxPos:=0;
	SysFileDelete(Logger_IndexFile);
	RETURN;
END_IF
(* Recover message data *)
hFile:=SysFileOpen(Logger_DataFile,'r');
IF hFile<>0 THEN
	SysFileSetPos(hFile,Logger.SendIdx);
	SysFileRead(hFile,ADR(Logger.SendData),Logger.SendLen);
	Logger.SendReq:=TRUE;
	SysFileClose(hFile);
END_IF
(* Clear index entry *)
hFile:=SysFileOpen(Logger_IndexFile,'a');
IF hFile<>0 THEN
	SysFileSetPos(hFile,pos);
	i:=0;
	SysFileWrite(hFile, ADR(i), 4);
	Logger.LastIdxPos:=SysFileGetPos(hFile);
	SysFileClose(hFile);
END_IF
END_ACTION
ACTION MsgSave:
(* Add log position in recovery indexes *)
hFile:=SysFileOpen(Logger_IndexFile,'a');
SysFileWrite(hFile, ADR(Logger.SendIdx), SIZEOF(Logger.SendIdx));
SysFileWrite(hFile, ADR(Logger.SendLen), SIZEOF(Logger.SendLen));
SysFileClose(hFile);
END_ACTION

(* POU Utils Functions/TCPCLIENT, ST *)
FUNCTION_BLOCK TCPCLIENT
(***********************************************************************************************************	*)
(* Version: 1.3b                        			          													*)
(* Date: 28.10.2014                   				          							            			*)
(***********************************************************************************************************	*)
(* WAGO Kontakttechnik GmbH Hansastr. 27 32423 Minden(Westf.)													*)
(* Tel. +0049 571/887-0 Fax. +0049 571/887-0																	*)
(* Author: VB																									*)
(***********************************************************************************************************	*)
(*Description:	A TCP client to read and write data with additional connection watchdog							*)
(*History:																										*)
(*Version 1.3b: 28.10.2014: Use DWORD address for IP (Andrea Ravasio)											*)
(*Version 1.3: 11.02.2011: Changes according to 750-880/881											 			*)
(*Version 1.2: 29.08.2007 Bugfix TCP Client																		*)
(*Version 1.1: 15.01.2007 Changes according to FW11																*)
(*Version 1.0: 09.03.2006 Release																				*)
(***********************************************************************************************************	*)
VAR CONSTANT
	STATE_CREATE     				 : BYTE:= 0;
	STATE_OPEN     					 : BYTE:= 1;
	STATE_IOCTL    					 : BYTE:= 2;
	STATE_CONNECT     				 : BYTE:= 10;
	STATE_TX       					 : BYTE:= 20;
	STATE_RX       					 : BYTE:= 30;
	STATE_CLOSE    					 : BYTE:= 40;
	STATE_ERROR_TRAP			     : BYTE:= 200;
END_VAR

VAR_INPUT
	xOpenConnection					: BOOL;
	dwInetAddr						: DWORD; (* <== Use SysSockInetAddr() value or
													swapped bytes order of SysSockGetHostByName() value *)
	wPortNumber						: WORD;
	ptSendData						: POINTER TO ARRAY[0..MAX_SEND_TCP_CLIENT] OF BYTE;
	diSendCount						: DINT;
	tConnectWatchdogTime		    : TIME := t#10s;
END_VAR
VAR_OUTPUT
	xConnected						: BOOL;
	diError 						: DINT := 0;
END_VAR
(* ErrorCodes -----------------------------------------
	16#8001 => No socket descriptor available 
	16#8002 => SysSockSend returns -1 
	16#8003 => Socket was "gracefully closed" 
	16#8004 => switching to none blocking mode fails
	16#8005 => SysSockClose() returns FALSE 
    16#8006 => SysSockConnect() fails
    16#8007 => SysSockSend() fails
	16#8008 => error state machine 
	16#8009 => timeout while waiting for data from server 
------------------------------------------------------------*)
VAR_IN_OUT
	xStartSend							: BOOL;
	aReceiveBuffer						: ARRAY [0..MAX_RECEIVE_TCP_CLIENT] OF BYTE;
	diReceiveCount						: DINT;
END_VAR
VAR
	m_State								: BYTE := 0;
	m_ReceiveBuffer						: ARRAY [0..MAX_RECEIVE_TCP_CLIENT_SOCKET] OF BYTE;
	m_Socket							: DINT;
	m_AddressInfo						: SOCKADDRESS;
	m_BytesReceived						: DINT;
	m_diReturn							: DINT;
	m_xReturn							: BOOL;
	m_IoCtlParameter  					: DINT := 1; (* IOCTL-Parameter for non-blocking mode of sockets *)
	i									: INT;
	T_Connect							: TON;
	m_count								: DINT;
	diOption							: DINT := 1;
	m_Blocking   						: DINT := 0;
END_VAR
IF xOpenConnection THEN
	(* State maschine *)
	CASE  m_State OF

	(* -------------------------------------------------------------------------*)
	STATE_CREATE:
			(* create socket descriptor*)
			m_Socket := SysSockCreate(diAddressFamily	:= SOCKET_AF_INET,
													 diType		:= SOCKET_STREAM,
													 diProtocol := SOCKET_IPPROTO_TCP);
			IF m_Socket >= 0 THEN
			(*Set Push-Bit*)
				IF ADR(%MW0)=16#30000000  OR ADR(%MW0)=16#20000000 THEN (*841 or 881*)
					SysSockSetOption(
						diSocket:=m_Socket,
						diLevel:=6,
						diOption:=SOCKET_TCP_NODELAY,
						pOptionValue:=ADR(diOption),
						diOptionLength:=SIZEOF(diOption));
				ELSE
						;
				END_IF
				m_State := STATE_IOCTL; (* succesful *)
			ELSE
				diError := 16#8001;  (* no socket descriptor available *)
				m_State := STATE_ERROR_TRAP;
			END_IF

	(* -------------------------------------------------------------------------*)
	STATE_IOCTL: (* change  socket mode  to none blocking *)
		m_diReturn := SysSockIoctl( m_Socket, SOCKET_FIONBIO, ADR(m_IoCtlParameter));
		IF m_diReturn <> 0 THEN
			m_AddressInfo.sin_family := SOCKET_AF_INET;
			m_AddressInfo.sin_port := SysSockNtohs(wPortNumber);
			m_AddressInfo.sin_addr := dwInetAddr;
			m_State := STATE_CONNECT;
		ELSE
			diError := 16#8004;  (* switching to none blocking mode fails *)
			m_State := STATE_ERROR_TRAP;
		END_IF


	(* -------------------------------------------------------------------------*)
	STATE_CONNECT: (* connect with server *)
		T_Connect(IN:=TRUE , PT:=tConnectWatchdogTime);(*activate watchdog for establishing connection to a server*)
		m_xReturn := SysSockConnect ( m_Socket, ADR(m_AddressInfo),  SIZEOF(m_AddressInfo));
		IF m_xReturn THEN (* succesful *)
			IF xStartSend THEN
				m_State := STATE_TX;(*transmit data*)
			ELSE
				m_State := STATE_RX;(*wait for data from server*)
			END_IF
			xConnected:=TRUE;
			T_Connect(IN:=FALSE);
		ELSE
			IF T_Connect.Q THEN
				diError := 16#8006;  (* connect fails *)
				xConnected:=FALSE;
				T_Connect(IN:=FALSE);
				m_State := STATE_ERROR_TRAP;
				SysSockClose( m_Socket);
			ELSE
				m_State := STATE_CONNECT;(*client still  tries to set up connection*)
			END_IF
		END_IF


	STATE_TX:	 (* send TCP-message *)
		m_diReturn := SysSockSend(diSocket := m_Socket,
								  pbyBuffer := ADR(ptSendData^[0]),
								  diBufferSize := diSendCount-m_count,
								  diFlags := 0);

		CASE m_diReturn OF
		-1:	(* ERROR *)
			T_Connect(IN:=TRUE , PT:=CONNECT_WATCHDOG_TIME);(*activate watchdog to check communication*)
			IF t_Connect.Q THEN
				diError := 16#8007;
				T_Connect(IN:=FALSE);
				m_State:=STATE_CLOSE;
			END_IF
		0: (* socket was "gracefully closed" *)
			m_State := STATE_CLOSE;
			diError := 16#8003;
		ELSE (* succesful *)
			m_count:=m_count+m_diReturn;
			IF m_count>=diSendCount THEN
				diError := 16#0000;
				m_State := STATE_RX;
				m_count:=0;
				xStartSend:=FALSE;
			END_IF
			T_Connect(IN:=FALSE);
		END_CASE

	(* -------------------------------------------------------------------------*)
	STATE_RX: (* process receive data *)
			m_BytesReceived := SysSockRecv(	diSocket 	:= m_Socket,
										pbyBuffer 	:= ADR(m_ReceiveBuffer),		(* Address of receive buffer *)
										diBufferSize:= SIZEOF(m_ReceiveBuffer),
										diFlags		:= 0);

			CASE m_BytesReceived OF
			-1:	(* No data available or error occured *)
				T_Connect(IN:=TRUE , PT:=tConnectWatchdogTime);(*activate watchdog to check communication*)
				IF t_Connect.Q THEN
					diError:=16#8009;
					T_Connect(IN:=FALSE);
					m_State:=STATE_CLOSE;
				END_IF
				IF xStartSend THEN
					m_State:=STATE_TX	;(* WAIT IN THIS STATE  and check for arriving data or new send command*)
				END_IF;
			0: (* socket was "gracefully closed"  *)
				m_State:=STATE_CLOSE;
				diError := 16#8003;
			ELSE (* succesful *)
				diError := 16#0000;
				T_Connect(IN:=FALSE);
				(* Copy received data into receive buffer *)
				FOR i:= 0 TO DINT_TO_INT(m_BytesReceived	)-1 DO
					aReceiveBuffer[diReceiveCount]:= m_ReceiveBuffer[i];
					diReceiveCount:=(diReceiveCount+1) MOD SIZEOF(aReceiveBuffer);
				END_FOR

			END_CASE

	(* -------------------------------------------------------------------------*)
	STATE_CLOSE : (* close socket *)
		IF ADR(%MW0)=16#30000000  OR ADR(%MW0)=16#20000000 THEN (*841 or 881*)
			;
		ELSE
			SysSockShutdown(m_Socket, 0);;(*870*)
		END_IF
		m_xReturn := SysSockClose( m_Socket);
		m_Socket := -1;
		m_State := 0; (* succesful *)
		xConnected:=FALSE;
		T_Connect(IN:=FALSE);
	(* -------------------------------------------------------------------------*)
	STATE_ERROR_TRAP: (* error handling *)
		xConnected:=FALSE;

	ELSE  (* Bad FSM code trap  *)
			m_State:= STATE_ERROR_TRAP;
			diError:= 16#8008;
	END_CASE

ELSE(*close connection*)
	IF m_Socket >= 0 THEN
		IF ADR(%MW0)=16#30000000  OR ADR(%MW0)=16#20000000 THEN (*841 or 881*)
			;
		ELSE
			SysSockShutdown(m_Socket, 0);;(*870*)
		END_IF
		SysSockClose( m_Socket);
	END_IF
	m_Socket := -1;
	diError := 16#0000;
	m_State := STATE_CREATE;
	xConnected:=FALSE;
	T_Connect(IN:=FALSE);
END_IF
END_FUNCTION_BLOCK

(* POU Utils Functions/DWORDSWAP, ST *)
FUNCTION DWORDSWAP:BOOL
VAR_INPUT
	pIn:POINTER TO ARRAY[1..4] OF BYTE;
	pOut:POINTER TO ARRAY[1..4] OF BYTE;
END_VAR
VAR
END_VAR
pOut^[1]:=pIn^[4];
pOut^[2]:=pIn^[3];
pOut^[3]:=pIn^[2];
pOut^[4]:=pIn^[1];
END_FUNCTION

(* POU Utils Functions/CHKSTRING, ST *)
FUNCTION CHKSTRING : BOOL
VAR_INPUT
	pString: POINTER TO BYTE;
	pPattern: POINTER TO BYTE;
END_VAR
VAR
END_VAR
CHKSTRING:=TRUE;
WHILE pPattern^<>0 AND CHKSTRING DO
	IF pPattern^<>pString^ THEN CHKSTRING:=FALSE; END_IF
	pString:=pString+1;
	pPattern:=pPattern+1;
END_WHILE
END_FUNCTION

(* POU TCP_Remote/Remote_Proc, ST *)
PROGRAM Remote_Proc
VAR
	s1:         	TCPSERVER;
	Enable: 		BOOL;
	Connected: 		BOOL;
	Error: 			DINT;

	TxData:			ARRAY [0..MAX_SEND_TCP_SERVER] OF BYTE;
	TxLen:			DINT;
	TxTrig:			BOOL;

	RxData:			ARRAY [0..MAX_RECEIVE_TCP_SERVER] OF BYTE;
	RxLen:			DINT;

	Status:			DINT;

	(* Command interpreter *)

	Cmd_Buf:		ARRAY [0..MAX_RECEIVE_TCP_SERVER] OF BYTE;
	Cmd_Buf_U16:	POINTER TO WORD;
	Cmd_Buf_INT:	POINTER TO INT;
	Cmd_BufLen:		WORD;
	Cmd_St:			WORD;

	Cmd_Obj:		WORD;
	Cmd_ObjIdx:		WORD;
	Cmd_C:			WORD;
	Cmd_R:			WORD;
	Cmd_CLen:		WORD;
	Cmd_RLen:		WORD;

	i : WORD;
	j : INT;
	s2 : STRING;

END_VAR
(*=== State machine ===*)
CASE Status OF
	0: (* Startup *)
		TxLen:=0; TxTrig:=FALSE;
		RxLen:=0;
		Enable:=TRUE;
		Status:=1;

	1: (* Wait incoming connection *)
		IF Connected THEN
			(* Log access *)(*
			LogEv(EL_Log,EO_VPN,1,5,'Remote');*)
			(* Send welcome message *)(*
			ADDSTRING(pTxData:=ADR(TxData), pString:=ADR(Remote_WELCOME), TxLen:=TxLen);
			TxTrig:=TRUE;*)
			(* Reset vars *)
			Cmd_BufLen:=0;
			Cmd_St:=0;
			Status:=2;
		END_IF
		IF Error>1 THEN
			Enable:=FALSE;
			Status:=0;
		END_IF

	2: (* Wait command *)
		IF RxLen>0 THEN
			(*=== Interpreter start ===*)
			IF Cmd_BufLen+(RxLen/2)>=MAX_RECEIVE_TCP_SERVER THEN
				(* ERROR *)
				Cmd_BufLen:=0;
			ELSE
				i:=HEXTORAW(pString:=ADR(RxData), StringLen:=DINT_TO_WORD(RxLen), pData:=ADR(Cmd_Buf[Cmd_BufLen]));
				Cmd_BufLen:=Cmd_BufLen+i;
			END_IF
			IF Cmd_BufLen>=8 THEN
				Cmd_Buf_U16:=ADR(Cmd_Buf[6]);
				IF Cmd_BufLen>=(8+Cmd_Buf_U16^) THEN
					Cmd_CLen:=Cmd_Buf_U16^;
					Cmd_Buf_U16:=ADR(Cmd_Buf[0]); Cmd_Obj:=Cmd_Buf_U16^;
					Cmd_Buf_U16:=ADR(Cmd_Buf[2]); Cmd_ObjIdx:=Cmd_Buf_U16^;
					Cmd_Buf_U16:=ADR(Cmd_Buf[4]); Cmd_C:=Cmd_Buf_U16^;
					(* Log command *)(*
					s2:='RCmd_';		s2:=CONCAT(s2,WORD_TO_STRING(Cmd_Obj));
					s2:=CONCAT(s2,'_'); s2:=CONCAT(s2,WORD_TO_STRING(Cmd_ObjIdx));
					s2:=CONCAT(s2,'_'); s2:=CONCAT(s2,WORD_TO_STRING(Cmd_C));
					s2:=CONCAT(s2,'_');	s2:=CONCAT(s2,WORD_TO_STRING(Cmd_CLen));
					LogEv(EL_Log,EO_VPN,1,6,s2);*)
					(* Execute command *)
					Command();
					Cmd_BufLen:=0;
				END_IF
			END_IF
			(*=== Interpreter end ===*)
			RxLen:=0;
		END_IF
		IF NOT Connected THEN
			Status:=0;
		END_IF

ELSE
	Status:=0;
END_CASE


(*=== Execute server lib ===*)
s1(
	xEnable				:= Enable,
	wPortNumber			:= Remote_PORT,
	tServerTimeOut		:= t#15m,
	ptSendData			:= ADR(TxData),
	diSendCount			:= TxLen,
	xStartSend			:= TxTrig,
	aReceiveBuffer		:= RxData,
	diReceiveCount		:= RxLen,
	xClientConnected	=> Connected,
	diError				=> Error
);
END_PROGRAM
ACTION Cmd_CAL:
(* Check index *)
(*IF Cmd_ObjIdx<>1 THEN
	Cmd_R:=2;
	RETURN;
END_IF

(* Process command *)
CASE Cmd_C OF

	1: (* GET CLIMATIC *)
		Cmd_RLen:=20;
		FOR i:=0 TO 4 DO
			j:=DINT_TO_INT(CAL01_Clima.Points[i].X);
			TxLen:=TxLen+RAWTOHEX(ADR(j),2,ADR(TxData[TxLen]));
			j:=DINT_TO_INT(CAL01_Clima.Points[i].Y);
			TxLen:=TxLen+RAWTOHEX(ADR(j),2,ADR(TxData[TxLen]));
		END_FOR

	2: (* SET CLIMATIC *)
		IF Cmd_CLen<>20 THEN
			Cmd_R:=4;
		ELSE
			FOR i:=0 TO 4 DO
				Cmd_Buf_INT:=ADR(Cmd_Buf[8+4*i]); j:=Cmd_Buf_INT^;
				CAL01_Clima.Points[i].X:=INT_TO_DINT(j);
				Cmd_Buf_INT:=ADR(Cmd_Buf[10+4*i]); j:=Cmd_Buf_INT^;
				CAL01_Clima.Points[i].Y:=INT_TO_DINT(j);
			END_FOR
		END_IF

ELSE
	Cmd_R:=3;
END_CASE*)
;
END_ACTION
ACTION Cmd_CRON:
(* Check index *)
IF Cmd_ObjIdx<1 OR Cmd_ObjIdx>9 THEN
	Cmd_R:=2;
	RETURN;
END_IF

(* Process command *)
CASE Cmd_C OF

